IF P2M2_MachCtrl.U.DT_iMode=1 THEN
	D_Sys.bP2M2Enable:=TRUE;	
ELSE
	D_Sys.bP2M2Enable:=FALSE;
END_IF

D_Sys.fM2MainSetPos:=arrAxis[P2M2_Axise.VirAxisName.VirMain].NcToPlc.ActPos;//2号叠片主虚轴位置 20240509 CF
D_Pro.bAn_M2LockReady:=P2M2_MachCtrl.An_b.GetPiceReady;//正极取流水线极片准备好
D_Pro.bAn_M2JumpReady:=P2M2_MachCtrl.An_b.JumpPiceReady  OR (bDiffVel[2] AND NOT P2M2_MachCtrl.An_b.GetPiceReady);//正极跳过取流水线极片准备好 20240509 CF
D_Pro.bCa_M2LockReady:=P2M2_MachCtrl.Ca_b.GetPiceReady;//负极取流水线极片准备好
D_Pro.bCa_M2JumpReady:=P2M2_MachCtrl.Ca_b.JumpPiceReady;//负极跳过取流水线极片准备好
D_Pro.bAn_M2PoleHave:=P2M2_MachCtrl.An_b.bAn_PoleHave;
D_Pro.bCa_M2PoleHave:=P2M2_MachCtrl.Ca_b.bCa_PoleHave;
//模切给叠片的信号
P2M2_MachCtrl.An_b.An_MainBeltOK:=M_Pro.bAn_M2Allow;//允许正极取极片
P2M2_MachCtrl.Ca_b.Ca_MainBeltOK:=M_Pro.bCa_M2Allow;//允许负极取极片



//运行时间统计
	DT2_Timedata(
							Alm:=P2M2_DTSysState.bErrorStop AND NOT P2M2_DError AND NOT P2M2_MachCtrl.DT_b.DT_GMchange(*OR  P2M2_WJSysState.bErrorStop*) , 
							Wait:=P2M2_MachCtrl.U.DT_iMode=3 AND NOT P2M2_MachCtrl.DT_b.DT_GMchange AND (NOT P2M2_DTSysState.bErrorStop OR P2M2_DError (*AND NOT  P2M2_WJSysState.bErrorStop*) )  , 
							Run:= P2M2_MachCtrl.U.DT_iMode=1 (*AND P2M2_MachCtrl.U.WJ_iMode=1 AND P2M2_MachCtrl.U.TJ_iMode=1*), 
							Overhang_NG:= P2M2_MachCtrl.DT_b.DT_OverhangNG, 
							GM_change:=P2M2_MachCtrl.DT_b.DT_GMchange , 
							Query:=P2M2_MachCtrl.DT_b.Query, 
							date1:=P2M2_MachCtrl.DT_b.date1 , 								
							STTimedata=> );

							
							
//隔膜物料码OK
IF  (P3_PLC_PC_MES.Mes_PcToPlc6 AND  LEN(P3_PLC_PC_MES.Station2_Code)>6  ) OR P2M2_MachCtrl.DT_b.PartNumberOff THEN
	P2M2_MachCtrl.DT_b.DiaphragmPartNumberOK:=TRUE;
ELSE
	P2M2_MachCtrl.DT_b.DiaphragmPartNumberOK:=FALSE;
END_IF
//蓝胶物料码OK
IF  (P3_PLC_PC_MES.Mes_PcToPlc9 AND  LEN(P3_PLC_PC_MES.Station2_BlueCode)>6  ) OR P2M2_MachCtrl.DT_b.PartNumberOff THEN
	P2M2_MachCtrl.DT_b.BluePartNumberOK:=TRUE;
ELSE
	P2M2_MachCtrl.DT_b.BluePartNumberOK:=FALSE;
END_IF



IF P2M2_MachCtrl.DT_b.DiaphragmPartNumberOK THEN//隔膜料号OK
	CellMemory[P2M2_MachCtrl.DT_b.DT_Memory].Station_Code :=P3_PLC_PC_MES.Station2_Code;	
ELSE
	CellMemory[P2M2_MachCtrl.DT_b.DT_Memory].Station_Code :='';	
END_IF
IF P2M2_MachCtrl.DT_b.BluePartNumberOK THEN//蓝胶料号OK
	CellMemory[P2M2_MachCtrl.DT_b.DT_Memory].Station_BlueCode :=P3_PLC_PC_MES.Station2_BlueCode;	
ELSE
	CellMemory[P2M2_MachCtrl.DT_b.DT_Memory].Station_BlueCode :='';	
END_IF


	
//物料码清理
//隔膜条码重新校验
DT2Code_MES[1](CLK:=arrCyCtrl[P2M2_CycNo.CylinderName.PoleInflationCy].Status.ONState  , Q=> );  
IF DT2Code_MES[1].Q THEN
	P2M2_MachCtrl.DT_b.DiaphragmPartNumberOK:=FALSE;
	P3_PLC_PC_MES.Station2_Code:='';
	P3_PLC_PC_MES.Mes_PcToPlc6:=FALSE;
END_IF	

//蓝胶条码重新校验						
DT2Code_MES[2](CLK:= P2M2_MachCtrl.DT_b.HMI_WinBtn[1] , Q=> );  
IF DT2Code_MES[2].Q THEN
	P2M2_MachCtrl.DT_b.BluePartNumberOK:=FALSE;
	P3_PLC_PC_MES.Station2_BlueCode:='';
	P3_PLC_PC_MES.Mes_PcToPlc9:=FALSE;
END_IF									

(*						
//物料码校验报警
IF NOT P2M2_MachCtrl.DT_b.DiaphragmPartNumberOK AND NOT P2M2_MachCtrl.DT_b.PartNumberOff THEN
	P2M2_MachCtrl.DT_b.Error[55]:=TRUE;//叠台隔膜物料码校验未通过，请重新校验物料码
END_IF
IF NOT P2M2_MachCtrl.DT_b.BluePartNumberOK AND NOT P2M2_MachCtrl.DT_b.PartNumberOff THEN
	P2M2_MachCtrl.DT_b.Error[56]:=TRUE;//叠台蓝胶物料码校验未通过，请重新校验物料码
END_IF							
*)							
							


IF P2Btn.P2M2_Autobtn THEN
    arrCyCtrl[163].Cmd.bOFF:=TRUE;	//2号叠台		隔膜接带平台除尘
    arrCyCtrl[163].Cmd.bON:=FALSE;
ELSE
   arrCyCtrl[163].Cmd.bON:=TRUE;
   arrCyCtrl[163].Cmd.bOFF:=FALSE;
END_IF

END_PROGRAM

// ---- P2POUs/POUS/P2M3_Auto.TcPOU
PROGRAM P2M3_Auto
VAR
	DT3Code_MES: ARRAY[1..10] OF R_TRIG;
END_VAR

// 3号叠台自动
P2M3_program(
	DTselect:=3 , 
	Sys_Control:=P2M3_sysControl , 
	Mach_Control:=P2M3_MachCtrl , 
	arrCyNo:=P2M3_CycNo , 
	AxiseNo:=P2M3_Axise ,
	TableNo:=P2M3_TableNo ,
	Par:=P2M3_Par ,
	CCD:=P2M3_CCD,
	Torque:=P2M3_Torque,
	iTargetTorqueTest=>iTargetTorque[3]);
	
	

//叠片给模切的信号
D_Pro.bAn_M3Done:=P2M3_MachCtrl.An_b.AN_BeltDone; //正极取流水线极片完成
D_Pro.bAn_M3Safety:=P2M3_MachCtrl.An_b.AN_BeltSafe;//正极取流水线安全位
D_Pro.bCa_M3Done:=P2M3_MachCtrl.Ca_b.Ca_BeltDone;//负极取水线极片完成
D_Pro.bCa_M3Safety:=P2M3_MachCtrl.Ca_b.Ca_BeltSafe;//负极取流水线安全位
//D_Sys.fM3MainSetPos:=arrAxisCtrl[VirAxisNo.P2M3_VirMain].Cmd.fSetPos;
//D_Sys.bP2M3Enable:=P2M3_MachCtrl.U.DT_ModelChees;

IF P2M3_MachCtrl.U.DT_iMode=1 THEN
	D_Sys.bP2M3Enable:=TRUE;	
ELSE
	D_Sys.bP2M3Enable:=FALSE;
END_IF


D_Sys.fM3MainSetPos:=arrAxis[P2M3_Axise.VirAxisName.VirMain].NcToPlc.SetPos;//3号叠片主虚轴位置 20240509 CF
D_Pro.bAn_M3LockReady:=P2M3_MachCtrl.An_b.GetPiceReady;//正极取流水线极片准备好
D_Pro.bAn_M3JumpReady:=P2M3_MachCtrl.An_b.JumpPiceReady  OR (bDiffVel[3] AND NOT P2M3_MachCtrl.An_b.GetPiceReady);//正极跳过取流水线极片准备好 20240509 CF
D_Pro.bCa_M3LockReady:=P2M3_MachCtrl.Ca_b.GetPiceReady;//负极取流水线极片准备好
D_Pro.bCa_M3JumpReady:=P2M3_MachCtrl.Ca_b.JumpPiceReady;//负极跳过取流水线极片准备好
D_Pro.bAn_M3PoleHave:=P2M3_MachCtrl.An_b.bAn_PoleHave;
D_Pro.bCa_M3PoleHave:=P2M3_MachCtrl.Ca_b.bCa_PoleHave;
//模切给叠片的信号
P2M3_MachCtrl.An_b.An_MainBeltOK:=M_Pro.bAn_M3Allow;//允许正极取极片
P2M3_MachCtrl.Ca_b.Ca_MainBeltOK:=M_Pro.bCa_M3Allow;//允许负极取极片


//运行时间统计
 DT3_Timedata(						
							Alm:=P2M3_DTSysState.bErrorStop AND NOT P2M3_DError AND NOT P2M3_MachCtrl.DT_b.DT_GMchange(*OR  P2M3_WJSysState.bErrorStop*) , 
							Wait:=P2M3_MachCtrl.U.DT_iMode=3 AND NOT P2M3_MachCtrl.DT_b.DT_GMchange AND (NOT P2M3_DTSysState.bErrorStop OR P2M3_DError (*AND NOT  P2M3_WJSysState.bErrorStop*) )  , 
							Run:= P2M3_MachCtrl.U.DT_iMode=1 (*AND P2M3_MachCtrl.U.WJ_iMode=1 AND P2M3_MachCtrl.U.TJ_iMode=1*), 
							Overhang_NG:= P2M3_MachCtrl.DT_b.DT_OverhangNG, 
							GM_change:=P2M3_MachCtrl.DT_b.DT_GMchange , 
							Query:=P2M3_MachCtrl.DT_b.Query, 
							date1:=P2M3_MachCtrl.DT_b.date1 , 								
							STTimedata=> );

							
//隔膜物料码OK
IF  (P3_PLC_PC_MES.Mes_PcToPlc7 AND  LEN(P3_PLC_PC_MES.Station3_Code)>6  ) OR P2M3_MachCtrl.DT_b.PartNumberOff THEN
	P2M3_MachCtrl.DT_b.DiaphragmPartNumberOK:=TRUE;
ELSE
	P2M3_MachCtrl.DT_b.DiaphragmPartNumberOK:=FALSE;
END_IF
//蓝胶物料码OK
IF  (P3_PLC_PC_MES.Mes_PcToPlc10 AND  LEN(P3_PLC_PC_MES.Station3_BlueCode)>6  ) OR P2M3_MachCtrl.DT_b.PartNumberOff THEN
	P2M3_MachCtrl.DT_b.BluePartNumberOK:=TRUE;
ELSE
	P2M3_MachCtrl.DT_b.BluePartNumberOK:=FALSE;
END_IF



IF P2M3_MachCtrl.DT_b.DiaphragmPartNumberOK THEN//隔膜料号OK
	CellMemory[P2M3_MachCtrl.DT_b.DT_Memory].Station_Code :=P3_PLC_PC_MES.Station3_Code;	
ELSE
	CellMemory[P2M3_MachCtrl.DT_b.DT_Memory].Station_Code :='';	
END_IF
IF P2M3_MachCtrl.DT_b.BluePartNumberOK THEN//蓝胶料号OK
	CellMemory[P2M3_MachCtrl.DT_b.DT_Memory].Station_BlueCode :=P3_PLC_PC_MES.Station3_BlueCode;	
ELSE
	CellMemory[P2M3_MachCtrl.DT_b.DT_Memory].Station_BlueCode :='';	
END_IF


	
//物料码清理
//隔膜条码重新校验
DT3Code_MES[1](CLK:=arrCyCtrl[P2M3_CycNo.CylinderName.PoleInflationCy].Status.ONState  , Q=> );  
IF DT3Code_MES[1].Q THEN
	P2M3_MachCtrl.DT_b.DiaphragmPartNumberOK:=FALSE;
	P3_PLC_PC_MES.Station3_Code:='';
	P3_PLC_PC_MES.Mes_PcToPlc7:=FALSE;
END_IF	
//蓝胶条码重新校验	
				
DT3Code_MES[2](CLK:= P2M3_MachCtrl.DT_b.HMI_WinBtn[1] , Q=> );  
IF DT3Code_MES[2].Q THEN
	P2M3_MachCtrl.DT_b.BluePartNumberOK:=FALSE;
	P3_PLC_PC_MES.Station3_BlueCode:='';
	P3_PLC_PC_MES.Mes_PcToPlc10:=FALSE;
END_IF					

(*
//物料码校验报警
IF NOT P2M3_MachCtrl.DT_b.DiaphragmPartNumberOK AND NOT P2M3_MachCtrl.DT_b.PartNumberOff THEN
	P2M3_MachCtrl.DT_b.Error[55]:=TRUE;//叠台隔膜物料码校验未通过，请重新校验物料码
END_IF
IF NOT P2M3_MachCtrl.DT_b.BluePartNumberOK AND NOT P2M3_MachCtrl.DT_b.PartNumberOff THEN
	P2M3_MachCtrl.DT_b.Error[56]:=TRUE;//叠台蓝胶物料码校验未通过，请重新校验物料码
END_IF							
*)		





IF P2Btn.P2M3_Autobtn THEN
    arrCyCtrl[194].Cmd.bOFF:=TRUE;	///3号叠台		隔膜接带平台除尘
    arrCyCtrl[194].Cmd.bON:=FALSE;
ELSE
   arrCyCtrl[194].Cmd.bON:=TRUE;
   arrCyCtrl[194].Cmd.bOFF:=FALSE;
END_IF

END_PROGRAM

// ---- P2POUs/POUS/MAIN.TcPOU
PROGRAM MAIN
VAR
	rt:ARRAY[1..10]OF R_TRIG;//上升沿触发
	ft:ARRAY[1..10]OF F_TRIG;//下升沿触发
	i:BYTE;
	bSave: BOOL;
	rt10: R_TRIG;
	bReadDataFirstCyle: BOOL;
	testii: INT;
	testii2: INT;
	bSaveDataTest: BOOL;
	bReadDataCyle2: BOOL;
	rtSaveData: R_TRIG;
	fbDataXML  :FB_DataXML; 	
	
	
	
	BUSY: BOOL;
	ERR: BOOL;
	ERRID: UDINT;
	CSData:    CS_Data;
	

	THNN: INT;
	MA100: BOOL;
	A1: BOOL;
	D1: BOOL;
	A2: BOOL;
	A3: BOOL;
	
	//iShort:        IShortTest;
	D2: INT;
	//stTime: TIMESTRUCT;
	strTime: STRING;
	BY1:  BYTE;
	AA1: BOOL;
	btest: BOOL;
	iPower: INT;
	iPowerSetp: INT;
	bytePower: BYTE:=16#01;
	boPower2: BOOL;
	k: INT:=1;
	PowerOnDone: BOOL;
   
	SJ0617: INT;
	tRead										:TON;
END_VAR

VAR
	bFirstCycle										        	:BOOL;	(*初始化用的*)
(*保存掉电保持参数*)
	FB_WritePersistentData1								: FB_WritePersistentData;
	tCycleTimer											: TON;
	bWrite												: BOOL;    (*定时自动保存*)
(*系统重启*)
	tNtDelayReset										:TON;
	bReboot											: BOOL;	(*重启系统的变量*)
	NT_Reboot1											: NT_Reboot;
(*系统关机*)
	NT_Shutdown1										: NT_Shutdown;
	tNtDelayShutdown									: TON;
	bShutdown											: BOOL;
(*远程桌面接管*)
	OpenRemoteDesktop									: NT_StartProcess;
	timerHMI											:TON;
(*系统时间获取*)
	NT_GetTime1											: NT_GetTime;
(*心跳信号*)
	bHeartBeat											:BOOL;
	tHeartBeatTime										:TIME:=t#0.5s;
	TonHeartBeat										:TON;

	TaskInfo											:	TaskInfoCtrl;
	loadParaStep: UINT;

    tonPowerOn  :Tc2_Standard.TON;
    tonPower       :Tc2_Standard.TON;


     STR1: STRING:='20200412160000';
	 STR2: STRING:='12345678ABCDE';
	 STR3: STRING:='SSDDFF1234  JJJJ';
	 size:UDINT;
END_VAR

(*===========================================版本号=================================================*)
//MachimeVersion:='V3.0-24/3/2';(*HMI显示当前程序版本号*)
IF versionwrite THEN
   MachimeVersion:=CONCAT(CONCAT(CONCAT(CONCAT('V',CONCAT( WORD_TO_STRING(stTime.wYear),'.')),WORD_TO_STRING(stTime.wMonth)),'.'),WORD_TO_STRING(stTime.wDay));
END_IF
(*
版本： 


(*
1、线扫OK与NG信号IO触发;（02.20）
2、叠台NG梯度踢废空叠隔膜程序；（02.20）
3、叠台NG梯度踢废下料方式程序；（02.20）
4、隔膜剩余长度计算程序;（02.21）
5、无极片编号传送带尾部排废程序；（02.23）
6、对齐度NG计数程序  （02.27）
7、接带后找极耳程序；（02.28）
8、模切风刀吹气程序；（3.2）
9、程序版本号程序；（3.2）
10、叠台搬运极耳真空检测程序；（3.3）
11、冷压扫二维码程序；（3.3）
12、隔膜剩余长度计算（通过卷径大小）程序;（03.3）
13、隔膜卷径报警值限定（93），卷径报警实时判断改为叠完一个电芯判断一次;（03.6）
14、叠台搬运和压刀凸轮曲线修改，压刀升降和压刀开合行程限定；（03.12）
15、模切线扫结果判定逻辑优化，线扫触发和结果计数；（03.12）
16、新增模切放卷尾料4连标程序；（03.13）
17、模切黄标和接带踢废程序优化；（03.13）
18、短卷针回零增加安全条件(短卷针旋转轴原点传感器需亮)；（03.13）
19、模切放卷激光器继电器控制启用；（3.17）
20、触摸屏门禁屏蔽取消；（3.17）
21、增加启动CCD自检弹窗，需要确认后才能启动；（3.26）
22、叠台气涨轴开关有信号，隔膜踢废；（3.26）
23、触摸屏三级权限；（3.26）
24、上位机优率表；（3.31）
25、黄标跳切计数；（3.26）
26、黄标计数；（4.1）
27、叠台增加调试模式；（4.2）
28、热切丝寿命计数；（4.2）
29、模切尾料四连标检测；（4.2）
30、对齐度单片踢废；（4.5）
31、隔膜尾料角度计算；（4.5）
32、断带后R角不冲切；（4.7）
33、黄标与接带感应后日志；（4.7）
34、极片间距报警；（4.17）
35、凸轮位置角度固定；（4.17）
36、空叠首尾层隔膜降速降张力；（4.17）
37、正极真空改成常开；（4.17）
38、纠偏台重复精度测试；（4.17）
39、二维码贴胶完成自动备胶默停、重胶；（4.20）
40、对齐度踢废后第一片纠偏平台不纠偏；（4.20）
41、叠台一键初始化；（4.20）
42、模切尺寸、倒装、分段皮带比例系数改成一致；（4.20）
43、尾卷纠偏到限位，凸轮耦合报警；（4.20）
44、叠最后一层隔膜负极叠台升降放片位置下降少一点；（4.20）
45、模切R角横深纵深闭环纠偏；（4.20）
46、CCD标定与重复精度测试电机到位后延时拍照；（4.20）
47、短卷针夹泄气真空；（4.21）
48、对齐度闭环纠偏；（4.21）
49、模切触发高速停止；（4.22）
50、叠片取分段皮带取料中信号提前复位；（4.22）
51、贴胶头进退增加软限位；（4.23）
52、叠台0步增加判断，正负极不能执行同时往叠台方向运动流程；（4.23）
53、热压一键初始化；（4.23）
*)
*)
(*====================================================================================================*)

TwinCAT_Nt();
IF tonPowerOn.ET>=T#1S THEN
     MAIN.RecipeData();
END_IF
IOLink();

tonPowerOn(IN:=PowerOnDone , PT:=T#15S , Q=> , ET=> );  //上电延时5S

IF tonPowerOn.Q AND fbDataXML.bReadParDone THEN
  MainState();
  FingerprintKey();  
  dDrauFan[1];// :=TRUE;
  dDrauFan[2];// :=TRUE;
ELSE
   Power();//接触器上电
END_IF
op();



SJ0617;


//字体设置成中文字体  解决了注释乱码的问题






// scRecipe(iRecipe2:=iRecipe );

ACTION op:
FOR i :=1 TO 50 DO
	IF Network1_OP[i] = 8 THEN
		bNetwork1_OP[i] := TRUE;
	ELSE
		bNetwork1_OP[i] := FALSE;
	END_IF
	
	IF Network2_OP[i] = 8 THEN
		bNetwork2_OP[i] := TRUE;
	ELSE
		bNetwork2_OP[i] := FALSE;
	END_IF
	
	IF Network3_OP[i] = 8 THEN
		bNetwork3_OP[i] := TRUE;
	ELSE
		bNetwork3_OP[i] := FALSE;
	END_IF
	
	IF Network4_OP[i] = 8 THEN
		bNetwork4_OP[i] := TRUE;
	ELSE
		bNetwork4_OP[i] := FALSE;
	END_IF
	
	IF Network5_OP[i] = 8 THEN
		bNetwork5_OP[i] := TRUE;
	ELSE
		bNetwork5_OP[i] := FALSE;
	END_IF
END_FOR
END_ACTION

ACTION Power:
(***系统延时启动***)

tonPower(IN:= , PT:=T#1.5S , Q=> , ET=> );

CASE iPowerSetp OF
0:
    tonPower.IN:=TRUE;
    iPowerSetp:=10;
10:
   IF   tonPower.Q  THEN
      bytePower:=SHL(bytePower,1);
     
      tonPower(IN:=FALSE );
      k:=k+1;
     iPowerSetp:=20;
  END_IF
20:
    bytePower.0:=1;
    tonPower.IN:=TRUE;
    iPowerSetp:=30;
30:
   IF  k>=8 THEN
        iPowerSetp:=666;
       // bytePower:=16#00;
        PowerOnDone:=TRUE;
   ELSE
      iPowerSetp:=10;
   END_IF

END_CASE
 
bytePower.0;
bytePower.1;
bytePower.2;
bytePower.3;
bytePower.4;
bytePower.5;
bytePower.6;
bytePower.7;
END_ACTION

ACTION RecipeData:

IF NOT  bReadDataFirstCyle AND tCycleTimer.ET>T#90S THEN //testii:=testii+1
	//fbDataXML.bRead:=NOT bDataValid;
	bReadDataFirstCyle:=TRUE;
END_IF


IF fbDataXML.bReadParDone AND bReadDataFirstCyle AND NOT  bReadDataCyle2 THEN
	  parDA:=P2User1_Par.parDA;
	  parFilterAD:=P2User1_Par.parFilterAD;//  先备份数据暂时不开放 
      bReadDataCyle2:=TRUE;
END_IF

rt[2](CLK:=tCycleTimer.ET>=T#4M , Q=> );
rtSaveData(CLK:=stHmiSysCmd.bSaveData , Q=> );
IF  rtSaveData.Q THEN
	bSaveDataTest:=TRUE;
END_IF
IF  rt[2].Q  OR  bSaveDataTest THEN   
	P2User1_Par.parDA:=parDA;
	P2User1_Par.parFilterAD:=parFilterAD; 
	bSaveDataTest:=FALSE;
	fbDataXML.bSave:=TRUE;
	testii2:=testii2+1;
END_IF

rt[4](CLK:=stHmiSysCmd.bReadData (*AND P2M1_MachCtrl.U.DT_iMode=3 AND P2M2_MachCtrl.U.DT_iMode=3 AND P2M3_MachCtrl.U.DT_iMode=3*), Q=> );
rt[5](CLK:=PowerOnDone , Q=> );
tRead(IN:=PowerOnDone, PT:=T#3S , Q=> , ET=> );
IF PowerOnDone AND  tRead.Q AND NOT fbDataXML.bReadParDone THEN
	 P2M3_MachCtrl.DT_b.Error[67]:=TRUE;//上电后叠台参数读取失败，请手动点读取参数
END_IF

fbDataXML(
					bSave:=fbDataXML.bSave AND NOT P2M3_MachCtrl.DT_b.Error[67] , 
					bRead:=fbDataXML.bRead OR rt[5].Q OR rt[4].Q , 
					bSaveParDone=> , 
					bReadParDone=> );

fbDataXML.bSaveParDone;
fbDataXML.bReadParDone;


(*
tCycleTimer(IN:=NOT tCycleTimer.Q , PT:=T#300S , Q=>bSave , ET=> );
rt10(clk:=bSave);
IF NOT  bReadDataFirstCyle THEN //testii:=testii+1
	 fbDataXML.bRead:=TRUE;
	 testii:=testii+1;
	 bReadDataFirstCyle:=TRUE;
END_IF


IF fbDataXML.bReadParDone AND bReadDataFirstCyle AND NOT  bReadDataCyle2 THEN
	  //parDA:=P2User1_Par.parDA;
	  //parFilterAD:=P2User1_Par.parFilterAD;      //  先备份数据暂时不开放 
      bReadDataCyle2:=TRUE;
END_IF


rtSaveData(CLK:=stHmiSysCmd.bSaveData , Q=> );
IF  rtSaveData.Q THEN
	bSaveDataTest:=TRUE;
END_IF


IF  rt10.Q   OR   bSaveDataTest THEN
   
     P2User1_Par.parDA:=parDA;
	 P2User1_Par.parFilterAD:=parFilterAD; 

    bSaveDataTest:=FALSE;

	fbDataXML.bSave:=TRUE;
	testii2:=testii2+1;
END_IF

fbDataXML(bSave:=fbDataXML.bSave AND M_Sys .P1SaveParDone , 
                      bRead:=fbDataXML.bRead AND M_Sys.P1ReadParDone ,
                      bSaveParDone=> , 
                      bReadParDone=>,);
(*
IF fbDataXML.bError THEN				  
		P3_Error[91]:=TRUE;	
END_IF			
*)	 					   
P2SaveParDone:=fbDataXML.bSaveParDone;
P2ReadParDone:=fbDataXML.bReadParDone;
*)
END_ACTION

ACTION TwinCAT_Nt:
//fPlcCycleTime_ms:=UDINT_TO_LREAL(_TaskInfo[0].CycleTime)/10000;

(***********************  保存掉电保持数据   **************************************)
tCycleTimer(IN:=NOT tCycleTimer.Q , PT:=T#386S , Q=>bWrite , ET=> );
rt[1](CLK:=tCycleTimer.ET>=T#3M, Q=>bWrite );
FB_WritePersistentData1(
	NETID:='' ,
	PORT:=852 ,
	START:=bWrite OR  stHmiSysCmd.bSaveData   ,//OR    _TaskInfo[1].FirstCycle
	TMOUT:=t#2s ,
	MODE:=SPDM_2PASS ,
	BUSY=>BUSY ,
	ERR=> ERR,
	ERRID=>ERRID );
ft[1](CLK:=BUSY , Q=> );
IF ft[1].Q THEN
	bDataValid:=TRUE;
END_IF	
	
(********************** 获取系统时间   ***************************************)
NT_GetTime1(
	NETID:='' ,
	START:=Pulse._1s.RT ,
	TMOUT:= ,
	BUSY=> ,
	ERR=> ,
	ERRID=> ,
	TIMESTR=>stTime );

	strTime:=CONCAT(CONCAT(CONCAT(CONCAT(CONCAT(CONCAT(CONCAT(CONCAT( CONCAT(CONCAT( WORD_TO_STRING(stTime.wYear),'-'), WORD_TO_STRING(stTime.wMonth)),'-'),WORD_TO_STRING(stTime.wDay)),
             '-'),WORD_TO_STRING(stTime.wHour)),'-'),WORD_TO_STRING(stTime.wMinute)),'-'),WORD_TO_STRING(stTime.wSecond));

(********************************** Systemfunctions **********************************************************)
	SysInfo(
		Reset				:= ,
		TimeStampTrig		:= Pulse._100ms.RT,
		//RunTimeNo			=> ,
		//ProjectName			=> ,
		//NumberOfTasks		=> ,
		//OnlineChangeCount	=> ,
		RetainVarErr		=> ,
		PersistenVarErr		=> ,
		TimeStampDT			=> ,
		TimeStamp			=> ,
		TimeStr				=> ,
		DateStr				=> ,
		TimeStamp2			=> ,
		TimeStruct			=> ,
		MonthDays			=> ,
		LeapYear			=> ,
		WeekOfYear			=> ,
		timezoneId			=>);

	TaskInfo(
		index				=> ,
		active				=> ,
		taskName			=> ,
		firstCycle			=> ,
		cycleTimeExceeded	=> ,
		cycleTime			=> ,
		lastExecTime		=> ,
		priority			=> ,
		cycleCount			=> );

	Pulse(
		BlinkSlow			=> ,
		Blink				=> ,
		BlinkFast			=> );	
		
	(*系统重启，CE远程桌面，系统时间，定时保存掉电数据，等系统常规动作*)
(**********************  通讯心跳信号   ***************************************)
TonHeartBeat(IN:=NOT TonHeartBeat.Q , PT:=tHeartBeatTime , Q=> , ET=> );
IF TonHeartBeat.Q THEN
	bHeartBeat:=NOT bHeartBeat;
END_IF

tNtDelayReset(IN:=stHmiSysCmd.bRebootPc OR bReboot , PT:=T#1S , Q=> , ET=> );
NT_Reboot1(
	NETID:='' ,
	DELAY:= ,
	START:=tNtDelayReset.Q  ,
	TMOUT:=DEFAULT_ADS_TIMEOUT ,
	BUSY=> ,
	ERR=> ,
	ERRID=> );

tNtDelayShutdown(IN:=stHmiSysCmd.bShutDownPc OR bShutDown , PT:=T#1S , Q=> , ET=> );	(*触摸屏上已经做了延时*)
NT_Shutdown1(
	NETID:= ,
	DELAY:= ,
	START:=tNtDelayShutdown.Q,
	TMOUT:=DEFAULT_ADS_TIMEOUT ,
	BUSY=> ,
	ERR=> ,
	ERRID=> );
END_ACTION

END_PROGRAM

// ---- P2POUs/BasicFunction/08_Data/FB_DataXML.TcPOU
FUNCTION_BLOCK FB_DataXML
VAR_INPUT
    	bSave:BOOL;
	    bRead:BOOL;
		bReadSel:BOOL;//参数读取选择，TRUE=选择恢复上电备份的参数
END_VAR
VAR_OUTPUT
    	bSaveParDone      :BOOL;
	    bReadParDone     :BOOL;
END_VAR

VAR
	iDataSetp: INT;
	i1: INT;
	i2:BYTE;
	rt100:Tc2_Standard.R_TRIG;
	rt101:Tc2_Standard.R_TRIG;
	rt102:Tc2_Standard.R_TRIG;
	rt103:Tc2_Standard.R_TRIG;
	bSaveTemp: BOOL;
	bReadTemp: BOOL;
	sFilePath:STRING;//文件路径
	sNewFilePath:STRING;//新文件路径
	sOldFilePath:STRING;//旧文件路径
	sFileName:STRING;//文件名称
	sVarName:STRING;//变量名称
	fbXmlSrvRead				: FB_XmlSrvReadByName;//读取XML文件	
	fbXmlSrvWrite				: FB_XmlSrvWriteByName;//写入XML文件
	bFirstCycleFlg:BOOL;//首次执行标志位
	fbGetFileList: FB_GetFileList;//获取文件列表功能块
	stFindFileEntry:ARRAY[1..50] OF ST_FindFileEntry;//文件列表存放结构体	
	nFileBakStep:UINT;//文件备份步序
	fbFileDelete	: FB_FileDelete;//删除文件
	fbFileRename	: FB_FileRename;//文件重命名
	fbCreateDirectory:FB_CreateDirectory;//文件夹创建
END_VAR

M_WriteOrRead();
A_FileBak();

ACTION A_FileBak:
CASE nFileBakStep OF
	200:
		fbGetFileList(bExecute:=FALSE);
		fbFileDelete(bExecute:=FALSE);
		fbFileRename(bExecute:=FALSE);
		fbCreateDirectory(bExecute:=FALSE);
		nFileBakStep:=300;
	300:(*获取文件列表*)
		fbGetFileList.pFindFileListADR:=ADR(stFindFileEntry);
		fbGetFileList.u32FindFileListSizeOf:=SIZEOF(stFindFileEntry);
		fbGetFileList(bExecute:=TRUE,sgPathName:=sOldFilePath,sgFileType:='xml');	
		IF fbGetFileList.bDone THEN
			fbGetFileList(bExecute:=FALSE);
			nFileBakStep:=310;
		ELSIF fbGetFileList.bError THEN
			fbGetFileList(bExecute:=FALSE);
			nFileBakStep:=997;
		END_IF
	310:(*判断文件是否存在，文件存在则备份一次，文件不存在直接给完成信号*)
		FOR i2:=1 TO 50 DO
			IF stFindFileEntry[i2].sFileName=sFileName THEN//
				EXIT;
			END_IF
		END_FOR
		IF i2>50 THEN
			nFileBakStep:=666;
		ELSE
			nFileBakStep:=320;
		END_IF
	320:(*文件夹创建*)
	fbCreateDirectory(bExecute:=TRUE , sgPathName:=sNewFilePath, tTimeout:=T#1S );
	IF fbCreateDirectory.bDone THEN
		fbCreateDirectory(bExecute:=FALSE);
		nFileBakStep:=350;
	ELSIF fbCreateDirectory.bError THEN
		fbCreateDirectory(bExecute:=FALSE);
		nFileBakStep:=998;
	END_IF
	350:(*删除旧文件*)
		fbFileDelete.sPathName:= CONCAT(sNewFilePath,sFileName);
		fbFileDelete(bExecute:=TRUE,ePath:= PATH_GENERIC,tTimeout:=T#5S);
		IF NOT fbFileDelete.bBusy THEN
			fbFileDelete(bExecute:=FALSE);
			nFileBakStep:=360;
		END_IF
	360:(*重命名文件*)
		fbFileRename.sOldName:= CONCAT(sOldFilePath,sFileName);
		fbFileRename.sNewName:= CONCAT(sNewFilePath,sFileName);
		fbFileRename(bExecute:=TRUE,ePath:= PATH_GENERIC,tTimeout:=T#5S);
		IF NOT fbFileRename.bBusy THEN
			fbFileRename(bExecute:=FALSE);
			IF NOT fbFileRename.bError THEN
				nFileBakStep:=666;
			ELSE
				nFileBakStep:=999;
			END_IF			
		END_IF
END_CASE
END_ACTION

ACTION M_WriteOrRead:
rt100(CLK:=bSave , Q=> );//保存参数
rt101(CLK:=bRead , Q=> );//读取参数
IF rt100.Q THEN  //保存参数
    bSaveTemp:=TRUE;
	bReadTemp:=FALSE;
	bSaveParDone:=FALSE;
	iDataSetp:=50;
END_IF
IF rt101.Q THEN  //读取参数
    bReadTemp:=TRUE;
    bSaveTemp:=FALSE;
	bReadParDone:=FALSE;
	iDataSetp:=50;
END_IF

//rt102(CLK:=NOT bFirstCycleFlg AND NOT bReadTemp, Q=> );//首次上电自动备份参数
IF rt102.Q THEN  //首次上电自动备份参数
	iDataSetp:=50;
END_IF

CASE  iDataSetp OF 
	50:
		I1:=1;
		fbXmlSrvRead(bExecute:=FALSE);
		fbXmlSrvWrite(bExecute:=FALSE);
		bSave:=FALSE;
		bRead:=FALSE;
		iDataSetp:=100;
	 100:
	 	sFilePath:='C:\P2XML\';//保存文件路径
		CASE I1 OF 
			1://轴参数
				sFileName  := 'P2arrAxisPar.xml';
				sVarName:='GMotion.arrAxisPar';
		(*		
			2://iModeEN
				sFileName  := 'P2iModeEN.xml';
				sVarName:='GVL_Par.iModeEN';
	     *)
			2://P2M1_Par
				sFileName  := 'P2M1_Par.xml';
				sVarName:='GVL_Par.P2M1_Par';
			3://P2M2_Par
				sFileName  := 'P2M2_Par.xml';
				sVarName:='GVL_Par.P2M2_Par';
			4: //P2M3_Par 
				sFileName  := 'P2M3_Par.xml';
				sVarName:='GVL_Par.P2M3_Par';
			5: // P2User1_Par
				sFileName  := 'P2User1_Par.xml';
				sVarName:='GVL_Par.P2User1_Par';
				
			(*	
			7: // P2M1_Production
				sFileName  := 'DT1Data.xml';
				sVarName:='GVL_Par.P2M1_Production';
			8: // P2M2_Production
				sFileName  := 'DT2Data.xml';
				sVarName:='GVL_Par.P2M2_Production';
			9: // P2M3_Production
				sFileName  := 'DT3Data.xml';
				sVarName:='GVL_Par.P2M3_Production';
		
			10: // P2User1_Par
				sFileName  := 'FilterAD.xml';
				sVarName:='GVL_Par.P2User1_Par';
			*)	
		END_CASE
		IF  bSaveTemp THEN
			iDataSetp:=200;
		ELSIF  bReadTemp THEN
			iDataSetp:=300;	
		//ELSIF NOT bFirstCycleFlg THEN
		//	iDataSetp:=400;
		END_IF
		
	(********************保存数据流程：先备份原来参数再保存新参数，如果保存失败恢复至备份参数********************)
	200:(*开始备份*)
		sNewFilePath:=CONCAT(sFilePath,'Tmp\');
		sOldFilePath:=sFilePath;
		nFileBakStep:=200;//调用A_FileBak()进行文件备份
		iDataSetp:=210;
	210:(*文件备份状态判断*)
		IF nFileBakStep=666 THEN//文件备份成功，保存新参数
			iDataSetp:=230;
		ELSIF nFileBakStep>990 THEN//文件备份失败
			iDataSetp:=997;			
		END_IF
	230:(*保存新参数*)	
		fbXmlSrvWrite(
			bExecute:= TRUE, 
			ePath:=PATH_GENERIC , 
			nMode:=XMLSRV_ADDMISSING , 
			sSymName:=sVarName , 
			sFilePath:= CONCAT(sFilePath,sFileName), 
			sXPath:= '/DataEntry/Value', 
			tTimeout:= T#2S);
		IF NOT fbXmlSrvWrite.bBusy THEN
			fbXmlSrvWrite(bExecute:=FALSE);
			IF NOT fbXmlSrvWrite.bError THEN(*保存新参数成功*)
				iDataSetp:=500;
			ELSE(*保存新参数失败，恢复未写入新参数前的备份*)
				iDataSetp:=250;
			END_IF	
		END_IF
	250:(*保存新参数失败，恢复未写入新参数前的备份*)
		sOldFilePath:=CONCAT('Tmp\' ,sFileName);
		sNewFilePath:=sFilePath;
		nFileBakStep:=200;//调用A_FileBak()进行文件备份
		iDataSetp:=260;
	260:(*恢复文件状态判断*)
		IF nFileBakStep=666 THEN//文件恢复成功
			iDataSetp:=500;
		ELSIF nFileBakStep>990 THEN//文件恢复失败
			iDataSetp:=998;			
		END_IF		

	(********************参数读取流程********************)	
	300:(*参数读取选择，TRUE=选择恢复上电备份的参数*)
		IF bReadSel THEN
			sFilePath:=CONCAT(sFilePath,'Bak\');
		END_IF
		iDataSetp:=310;
	310:(*读取参数*)
		fbXmlSrvRead(
			bExecute:= TRUE, 
			ePath:=PATH_GENERIC , 
			nMode:=XMLSRV_ADDMISSING , 
			sSymName:= sVarName, 
			sFilePath:=CONCAT(sFilePath,sFileName) , 
			sXPath:='/DataEntry/Value' , 
			tTimeout:=T#2S);
		IF NOT fbXmlSrvRead.bBusy THEN
			fbXmlSrvRead(bExecute:=FALSE);
			IF NOT fbXmlSrvRead.bError THEN
				iDataSetp:=500;//读取成功
			ELSE
				iDataSetp:=999;//读取失败
			END_IF
		END_IF
		
	(********************上电自动备份流程，防止被覆盖********************)	
	400:
		sOldFilePath:=sFilePath;
		sNewFilePath:=CONCAT(sFilePath,'Bak\' );
		nFileBakStep:=200;//调用A_FileBak()进行文件备份
		iDataSetp:=410;
	410:
		IF nFileBakStep=666 THEN
				iDataSetp:=500;
		ELSIF nFileBakStep>990 THEN
				iDataSetp:=999;			
		END_IF
	500:(*继续写下个文件*)
		IF 1<=i1 AND i1<5 THEN
			i1:=i1+1; 
			iDataSetp:=100; 
		ELSIF i1>=5 THEN
			IF  bSaveTemp THEN		
				bSaveParDone:=TRUE;
			ELSIF  bReadTemp THEN
				bReadParDone:=TRUE;
			ELSIF NOT bFirstCycleFlg THEN
				bFirstCycleFlg:=TRUE;
			END_IF
			bReadSel:=FALSE;
			bReadTemp:=FALSE;
			bSaveTemp:=FALSE;
			iDataSetp:=666;   
		END_IF
END_CASE
END_ACTION

END_FUNCTION_BLOCK

// ---- P2POUs/BasicFunction/08_Data/CS_Data.TcPOU
FUNCTION_BLOCK CS_Data
VAR_INPUT
END_VAR
VAR_OUTPUT
END_VAR
VAR
	//tDataSave:TON;
	//fbSaveData:FB_WritePersistentData;
	//fbXMLWrite:FB_XMLSrvWrite;
	//bWriteXml: BOOL;
	
	fbFileOpen_w:fb_fileopen;
	//fbFileOpen_r:fb_fileopen;
	fbFileWrite:fb_filewrite;
	fbFileRead:FB_FileRead;
	fbFileClose_w:fb_FileClose;
	//fbFileClose_r:fb_FileClose;
	HFILE:UINT;
	//HFILE_R:UINT;
	//bFileOpen_w:BOOL;
	//bFileOpen_r:BOOL;
	//bFileWrite:BOOL;
	//bFileClose_w:BOOL;
	//bFileClose_r:BOOL;
	//bFileRead:BOOL;
	bSave:BOOL;
	bRead:BOOL;
//	tFileOper_Save:TON;
	//tFileOper_Read:TON;
	iDataSetp: INT;
	TON10:Tc2_Standard.TON;
	bExecute: BOOL;
	I1: INT;
	rt100:Tc2_Standard.R_TRIG;
	rt101:Tc2_Standard.R_TRIG;
	bExecute1: BOOL;
	bExecute2: BOOL;
	bExecute3: BOOL;	

	bSaveTemp: BOOL;
	bReadTemp: BOOL;
	bReadDataOk: BOOL;
END_VAR


M_WriteOrRead();

ACTION M_WriteOrRead:


(*
rt100(CLK:=bSave , Q=> );//保存参数
rt101(CLK:=bRead , Q=> );//读取参数

IF rt100.Q THEN
	iDataSetp:=100;
	TON10.IN:=FALSE;
	I1:=1;
	bExecute1:=FALSE;
	bExecute2:=FALSE;	
	bExecute3:=FALSE;	
	bSave:=FALSE;
	bRead:=FALSE;
    bSaveTemp:=TRUE;
	bReadTemp:=FALSE;
END_IF

IF rt101.Q THEN
	iDataSetp:=100;
	TON10.IN:=FALSE;
	I1:=1;
	bExecute1:=FALSE;
	bExecute2:=FALSE;	
	bExecute3:=FALSE;	
	bSave:=FALSE;
	bRead:=FALSE;
    bReadTemp:=TRUE;
    bSaveTemp:=FALSE;
END_IF

TON10(IN:= , PT:=T#200MS , Q=> , ET=> );
//保存配方	
CASE  iDataSetp OF 
	
	100:	//参数给定
	   
	   IF bSaveTemp THEN
	     fbFileOpen_w.nMode:=FOPEN_MODEWRITE OR FOPEN_MODEBINARY;
	   END_IF
	   IF bReadTemp THEN
	     fbFileOpen_w.nMode:=FOPEN_MODEREAD OR  FOPEN_MODEBINARY;
	   END_IF
	  iDataSetp:=101;
	101:

	  CASE I1 OF 
		1:
		 fbFileWrite.pWriteBuff:=ADR(gstM1Par);
		 fbFileWrite.cbWriteLen:=SIZEOF(gstM1Par);
		 fbFileRead.pReadBuff:=ADR(gstM1Par1);
		 fbFileRead.cbReadLen:=SIZEOF(gstM1Par1);
		 fbFileOpen_w.sPathName:='C:\P2Data\M1.bin';
		2:
		 fbFileWrite.pWriteBuff:=ADR(gstM2Par);
		 fbFileWrite.cbWriteLen:=SIZEOF(gstM2Par);
		 fbFileRead.pReadBuff:=ADR(gstM2Par1);
		 fbFileRead.cbReadLen:=SIZEOF(gstM2Par1);
		 fbFileOpen_w.sPathName:='C:\P2Data\M2.bin';
		3:
		 fbFileWrite.pWriteBuff:=ADR(gstM3Par);
		 fbFileWrite.cbWriteLen:=SIZEOF(gstM3Par);
		 fbFileRead.pReadBuff:=ADR(gstM3Par1);
		 fbFileRead.cbReadLen:=SIZEOF(gstM3Par1);
		 fbFileOpen_w.sPathName:='C:\P2Data\M3.bin';
		4:
		 fbFileWrite.pWriteBuff:=ADR(gstM4Par);
		 fbFileWrite.cbWriteLen:=SIZEOF(gstM4Par);
		 fbFileRead.pReadBuff:=ADR(gstM4Par1);
		 fbFileRead.cbReadLen:=SIZEOF(gstM4Par1);
		 fbFileOpen_w.sPathName:='C:\P2Data\M4.bin';
		5:  
		 fbFileWrite.pWriteBuff:=ADR(gstM5Par);
		 fbFileWrite.cbWriteLen:=SIZEOF(gstM5Par); 
		 fbFileRead.pReadBuff:=ADR(gstM5Par1);
		 fbFileRead.cbReadLen:=SIZEOF(gstM5Par1);
		 fbFileOpen_w.sPathName:='C:\P2Data\M5.bin';
	  END_CASE
	  iDataSetp:=200;
	
	200:	//打开文件
		bExecute1:=TRUE;
		TON10.IN:=TRUE;
	  IF TON10.Q THEN
		 bExecute1:=FALSE; 
		 TON10.IN:=FALSE;
		 iDataSetp:=300; 
	  END_IF
	
	300:	//读写文件
		bExecute2:=TRUE;
		TON10.IN:=TRUE;
	  IF TON10.Q THEN
		  bExecute2:=FALSE; 
		  TON10.IN:=FALSE;
		 iDataSetp:=400; 
	  END_IF
	
	400:	//关闭文件
		bExecute3:=TRUE;
		TON10.IN:=TRUE;
	  IF TON10.Q THEN
		  bExecute3:=FALSE; 
		  TON10.IN:=FALSE;
		  iDataSetp:=500; 
	  END_IF
	
	500://继续写下个文件
	  IF I1>=1 AND I1<5 THEN
		 I1:=I1+1; 
		 TON10.IN:=FALSE;
		 iDataSetp:=100; 
		 bExecute1:=FALSE; 
		 bExecute2:=FALSE; 
		 bExecute3:=FALSE; 
	  ELSIF I1>=5 THEN
		  bReadTemp:=FALSE;
          bSaveTemp:=FALSE;
		 iDataSetp:=666;   
	  END_IF
END_CASE


IF bReadDataOk THEN
   gstM1Par:=gstM1Par1;
   gstM2Par:=gstM2Par1;
   gstM3Par:=gstM3Par1;
   gstM4Par:=gstM4Par1;	
   gstM5Par:=gstM5Par1;
   bReadDataOk:=FALSE;
END_IF










   	fbFileOpen_w(
	sNetId:= , 
	sPathName:= , //C:\P2Data
	nMode:=   , 
	ePath:=PATH_GENERIC , 
	bExecute:=bExecute1 , 
	tTimeout:=T#3S , 
	bBusy=> , 
	bError=> , 
	nErrId=> , 
	hFile=>hfile );


	fbFileWrite(
	sNetId:= , 
	hFile:= hFile, 
	pWriteBuff:= , 
	cbWriteLen:= , 
	bExecute:=bExecute2 AND bSaveTemp, 
	tTimeout:=T#3S , 
	bBusy=> , 
	bError=> , 
	nErrId=> , 
	cbWrite=> );



	fbFileRead(
	sNetId:= , 
	hFile:=hFile , 
	pReadBuff:= , 
	cbReadLen:= , 
	bExecute:= bExecute2 AND bReadTemp, 
	tTimeout:= T#3S, 
	bBusy=> , 
	bError=> , 
	nErrId=> , 
	cbRead=> , 
	bEOF=> );


	fbFileClose_w(
	sNetId:= , 
	hFile:= hFile, 
	bExecute:= bExecute3, 
	tTimeout:=T#3S , 
	bBusy=> , 
	bError=> , 
	nErrId=> );
	
	
	
*)
END_ACTION

END_FUNCTION_BLOCK

// ---- P2POUs/BasicFunction/11_SystemInfo/TaskInfoCtrl.TcPOU
FUNCTION_BLOCK TaskInfoCtrl
VAR_INPUT
END_VAR
VAR_OUTPUT
	index						:	INT;
	active					:	BOOL; 		(* Diese Variable zeigt an, ob die Task aktiv ist.*)
	taskName					:	STRING(16);	(* Der Taskname.*)
	firstCycle				:	BOOL;			(* Diese Variable hat im ersten Zyklus der SPS-Task den Wert: TRUE.*)
	cycleTimeExceeded		:	BOOL;			(* In dieser Variablen wird ein 躡erschreiten der eingestellten Taskzykluszeit gemeldet*)
	cycleTime				:	UDINT;		(* Eingestellte Taskzykluszeit in Vielfachen von 100ns*)
	lastExecTime			:	UDINT;		(* Ben鰐igte Zykluszeit f黵 den letzten Zyklus in Vielfachen von 100 ns*)
	MaxExecTime				:	UDINT;		(* Maximale Zykluszeit *)
	priority					:	BYTE;			(* Eingestellte Prioritaet der Task*)
	cycleCount				: 	UDINT;		(* Zykluszaehler*)
END_VAR

VAR
	GETCURTASKINDEX		: GETCURTASKINDEX;
END_VAR

	(*********************************************************************************)
	(*	(c) by Beckhoff Automation																		*)
	(*																											*)
	(*		B E C K H O F F   N E W   A U T O M A T I O N   T E C H N O L O G Y        *)
	(*																											*)
	(*		Eiserstr.5	D-33415 Verl	Germany	phone:	+49-5246-0	www.Beckhoff.com	*)
   (*																											*)
   (*		Bausteinbeschreibung	: Auswerten des SystemInfoTaskArrays 						*)
	(*																											*)
	(*		Version				:	V1.0																	*)
	(*		Stand					:	04.2009																*)
 	(*		Autor					:	Daniel Schlingmann												*)
	(*																											*)
	(*********************************************************************************)

(* Get Current Task Index ************************************************************************)
	GETCURTASKINDEX(index => index);

	(* Retein/Persisten Data Err *)
	//active :=  _TaskInfo[index].active;
	taskName :=  _TaskInfo[index].TaskName;
	firstCycle :=  _TaskInfo[index].FirstCycle;
	cycleTimeExceeded :=  _TaskInfo[index].CycleTimeExceeded;
	cycleTime :=  _TaskInfo[index].CycleTime;
	lastExecTime :=  _TaskInfo[index].LastExecTime;
	MaxExecTime	:= MAX(lastExecTime,MaxExecTime);
//	priority :=  _TaskInfo[index].Priority;
	firstCycle :=  _TaskInfo[index].FirstCycle;
	cycleCount :=  _TaskInfo[index].CycleCount;

(**************************************************************************************************)

END_FUNCTION_BLOCK

// ---- P2POUs/POUS/IOLink.TcPOU
PROGRAM IOLink
VAR
//	tFlash: TON;
//	bFlash:BOOL;
//	bIOinit: BOOL;
	XXX: INT;
	Q20815: BOOL;
	AA: INT;

     arrFilter_AD               : ARRAY[1..MaxAINo]  OF  FB_Filter_AD ;
      arrFilter_ADV2               : ARRAY[1..3]  OF  FB_Filter_ADV2 ;


    Test:BOOL;
	I1: INT;

    rt01   :Tc2_Standard.R_TRIG;
    rt02   :Tc2_Standard.R_TRIG;

     parDAOld                   :ARRAY[1..44] OF INT;   
	 q:INT;


END_VAR

P2_InPut();

P2_OutPut();

AI();

//LimitSwitch();

P2_AutoLink();
P2M1_AutoLink();
P2M2_AutoLink();
P2M3_AutoLink();
LimitSwitch();


IF fbPulseCtrl[4].RT THEN
      AO();
END_IF
(*
//rt01(CLK:=arrCyCtrl[P3CYNo.RollPress].Cmd.bON , Q=> );
//rt02(CLK:=arrCyCtrl[P3CYNo.RollPress].Cmd.bOFF , Q=> );
IF rt01.Q THEN
    P3EL4004S[3,1]:=parDA[33]	 ;//重力补偿
  //  P3EL4004S[3,2]:=parDA[34]	 ;
END_IF
IF rt02.Q THEN
    P3EL4004S[3,1]:=22000;//重力补偿
 //   P3EL4004S[3,2]:=20000;
END_IF



*)





AA;

ACTION AI:
//1号叠片
arrFilter_AD[1].AD	:=AI30[1];	//1号叠片	隔膜卷径超声波检测
arrFilter_AD[1].iMode:=2;
arrFilter_AD[1].fPointNum:=20;

arrFilter_AD[2].AD	:=AI30[2];	//1号叠片	隔膜放卷纠偏前检测
arrFilter_AD[2].iMode:=2;
arrFilter_AD[2].fPointNum:=20;//30;

arrFilter_AD[3].AD	:=AI30[3];	//1号叠片	隔膜放卷纠偏后检测
arrFilter_AD[3].iMode:=2;
arrFilter_AD[3].fPointNum:=20;//30;

//arrFilter_AD[4].AD	:=AI30[4];//1号叠片	隔膜张力检测
arrFilter_ADV2[1].AD	:=AI30[4];//1号叠片	隔膜张力检测
arrFilter_ADV2[1].iMode:=2;
arrFilter_ADV2[1].fPointNum:=1000;
//2号叠片
arrFilter_AD[5].AD	:=ABS(AI40[1]);	//2号叠片	隔膜卷径超声波检测
arrFilter_AD[5].iMode:=2;
arrFilter_AD[5].fPointNum:=20;

arrFilter_AD[6].AD	:=ABS(AI40[2]);	//2号叠片	隔膜放卷纠偏前检测
arrFilter_AD[6].iMode:=2;
arrFilter_AD[6].fPointNum:=20;//30;

arrFilter_AD[7].AD	:=ABS(AI40[3]);	//2号叠片	隔膜放卷纠偏后检测
arrFilter_AD[7].iMode:=2;
arrFilter_AD[7].fPointNum:=20;//30;

//arrFilter_AD[8].AD	:=ABS(AI40[4]);//2号叠片	隔膜张力检测
arrFilter_ADV2[2].AD	:=ABS(AI40[4]);//2号叠片	隔膜张力检测
arrFilter_ADV2[2].iMode:=2;
arrFilter_ADV2[2].fPointNum:=1000;
//3号叠片
arrFilter_AD[9].AD	:=ABS(AI50[1]);	//3号叠片	隔膜卷径超声波检测
arrFilter_AD[9].iMode:=2;
arrFilter_AD[9].fPointNum:=20;

arrFilter_AD[10].AD	:=ABS(AI50[2]);	//3号叠片	隔膜放卷纠偏前检测
arrFilter_AD[10].iMode:=2;
arrFilter_AD[10].fPointNum:=20;//30;

arrFilter_AD[11].AD	:=ABS(AI50[3]);	//3号叠片	隔膜放卷纠偏后检测
arrFilter_AD[11].iMode:=2;
arrFilter_AD[11].fPointNum:=20;//30;

//arrFilter_AD[12].AD	:=ABS(AI50[4]);//3号叠片	隔膜张力检测
arrFilter_ADV2[3].AD	:=ABS(AI50[4]);//3号叠片	隔膜张力检测
arrFilter_ADV2[3].iMode:=2;
arrFilter_ADV2[3].fPointNum:=1000;

FOR  I1:=1 TO  12  DO//MaxAINo
	IF  I1=4  THEN
           arrFilter_ADV2[1](
			  iMode:=         , 
			  AD:=				arrFilter_ADV2[1].AD, 
			  iLimitH:=         parFilterAD[4].iLimitH  , 
			  iLimitL:=          parFilterAD[4].iLimitL   , 
			  fRangeH:=      parFilterAD[4].fRangeH , 
			  fRangeL:=       parFilterAD[4].fRangeL , 
			  fPointNum:=    , 
			  Out_Value=>    );
  ELSIF  I1=8 THEN
           arrFilter_ADV2[2](
			  iMode:=         , 
			  AD:=			    arrFilter_ADV2[2].AD, 
			  iLimitH:=         parFilterAD[8].iLimitH  , 
			  iLimitL:=          parFilterAD[8].iLimitL   , 
			  fRangeH:=      parFilterAD[8].fRangeH , 
			  fRangeL:=       parFilterAD[8].fRangeL , 
			  fPointNum:=    , 
			  Out_Value=>);
  ELSIF  I1=12 THEN
           arrFilter_ADV2[3](
			  iMode:=         , 
			  AD:=				arrFilter_ADV2[3].AD, 
			  iLimitH:=         parFilterAD[12].iLimitH  , 
			  iLimitL:=          parFilterAD[12].iLimitL   , 
			  fRangeH:=      parFilterAD[12].fRangeH , 
			  fRangeL:=       parFilterAD[12].fRangeL , 
			  fPointNum:=    , 
			  Out_Value=>);
ELSE
	  arrFilter_AD[I1](
		  iMode:=         , 
		  AD:=				arrFilter_AD[I1].AD               , 
		  iLimitH:=         parFilterAD[I1].iLimitH  , 
		  iLimitL:=          parFilterAD[I1].iLimitL   , 
		  fRangeH:=      parFilterAD[I1].fRangeH , 
		  fRangeL:=       parFilterAD[I1].fRangeL , 
		  fPointNum:=    , 
		  Out_Value=>);
END_IF

END_FOR
//一号叠台
//P2M1_MachCtrl.DT_b.fWindDiameter:=arrFilter_AD[1].Out_Value;
P2M1_MachCtrl.DT_b.RecDevPV:=arrFilter_AD[2].Out_Value;
P2M1_MachCtrl.DT_b.RecDevPV1:=arrFilter_AD[3].Out_Value;
P2M1_MachCtrl.DT_b.TenAnglePos:=LREAL_TO_REAL(arrAxis[P2M1_Axise.AxisName.SEPTATension].NcToPlc.ActPos);	
P2M1_Par.stDT_date.fRectifyMaxValue:= parFilterAD[2].fRangeH;
P2M1_Par.stDT_date.fRectifyMinValue:=parFilterAD[2].fRangeL;
arrFilter_ADV2[1].Out_Value;

//二号叠台
//P2M2_MachCtrl.DT_b.fWindDiameter:=arrFilter_AD[5].Out_Value;
P2M2_MachCtrl.DT_b.RecDevPV:=arrFilter_AD[6].Out_Value;
P2M2_MachCtrl.DT_b.RecDevPV1:=arrFilter_AD[7].Out_Value;
P2M2_MachCtrl.DT_b.TenAnglePos:=LREAL_TO_REAL(arrAxis[P2M2_Axise.AxisName.SEPTATension].NcToPlc.ActPos);	//2号叠片	隔膜张力检测;
P2M2_Par.stDT_date.fRectifyMaxValue:= parFilterAD[6].fRangeH;
P2M2_Par.stDT_date.fRectifyMinValue:=parFilterAD[6].fRangeL;
arrFilter_ADV2[2].Out_Value;
//三号叠台
//P2M3_MachCtrl.DT_b.fWindDiameter:=arrFilter_AD[9].Out_Value;
P2M3_MachCtrl.DT_b.RecDevPV:=arrFilter_AD[10].Out_Value;
P2M3_MachCtrl.DT_b.RecDevPV1:=arrFilter_AD[11].Out_Value;
P2M3_MachCtrl.DT_b.TenAnglePos:=LREAL_TO_REAL(arrAxis[P2M3_Axise.AxisName.SEPTATension].NcToPlc.ActPos);	//3号叠片	隔膜张力检测
P2M3_Par.stDT_date.fRectifyMaxValue:= parFilterAD[10].fRangeH;
P2M3_Par.stDT_date.fRectifyMinValue:=parFilterAD[10].fRangeL;
arrFilter_ADV2[3].Out_Value;
END_ACTION

ACTION AO:
;
END_ACTION

ACTION LimitSwitch:

//1号叠台
arrAxisCtrl[P2AxisNo.P2M1_AnCarryingLine].Io.DigitalInputs;//一号叠台正极搬运平移//直线电机
arrAxisCtrl[P2AxisNo.P2M1_AnCarryingLine].Io.biPosLimit:= arrAxisCtrl[P2AxisNo.P2M1_AnCarryingLine].Io.DigitalInputs.17;
arrAxisCtrl[P2AxisNo.P2M1_AnCarryingLine].Io.biNegLimit:=  arrAxisCtrl[P2AxisNo.P2M1_AnCarryingLine].Io.DigitalInputs.18;
arrAxisCtrl[P2AxisNo.P2M1_AnCarryingLine].Io.biHomeSwitch:=arrAxisCtrl[P2AxisNo.P2M1_AnCarryingLine].Io.DigitalInputs.20;

arrAxisCtrl[P2AxisNo.P2M1_AnCarryingUpDown].Io.DigitalInputs;//一号叠台正极送片搬运升降
arrAxisCtrl[P2AxisNo.P2M1_AnCarryingUpDown].Io.biPosLimit:= arrAxisCtrl[P2AxisNo.P2M1_AnCarryingUpDown].Io.DigitalInputs.16;
arrAxisCtrl[P2AxisNo.P2M1_AnCarryingUpDown].Io.biNegLimit:=  arrAxisCtrl[P2AxisNo.P2M1_AnCarryingUpDown].Io.DigitalInputs.2;
arrAxisCtrl[P2AxisNo.P2M1_AnCarryingUpDown].Io.biHomeSwitch:=arrAxisCtrl[P2AxisNo.P2M1_AnCarryingUpDown].Io.DigitalInputs.2;

arrAxisCtrl[P2AxisNo.P2M1_AnCarryingWhirling].Io.DigitalInputs;//一号叠台正极搬运旋转
arrAxisCtrl[P2AxisNo.P2M1_AnCarryingWhirling].Io.biPosLimit:= arrAxisCtrl[P2AxisNo.P2M1_AnCarryingWhirling].Io.DigitalInputs.16;
arrAxisCtrl[P2AxisNo.P2M1_AnCarryingWhirling].Io.biNegLimit:=  arrAxisCtrl[P2AxisNo.P2M1_AnCarryingWhirling].Io.DigitalInputs.2;
arrAxisCtrl[P2AxisNo.P2M1_AnCarryingWhirling].Io.biHomeSwitch:=arrAxisCtrl[P2AxisNo.P2M1_AnCarryingWhirling].Io.DigitalInputs.2;

arrAxisCtrl[P2AxisNo.P2M1_AndeviationX1].Io.DigitalInputs;//一号叠台正极纠偏平台X1
arrAxisCtrl[P2AxisNo.P2M1_AndeviationX1].Io.biPosLimit:= arrAxisCtrl[P2AxisNo.P2M1_AndeviationX1].Io.DigitalInputs.16;
arrAxisCtrl[P2AxisNo.P2M1_AndeviationX1].Io.biNegLimit:=  arrAxisCtrl[P2AxisNo.P2M1_AndeviationX1].Io.DigitalInputs.17;
arrAxisCtrl[P2AxisNo.P2M1_AndeviationX1].Io.biHomeSwitch:=arrAxisCtrl[P2AxisNo.P2M1_AndeviationX1].Io.DigitalInputs.2;

arrAxisCtrl[P2AxisNo.P2M1_AndeviationX2].Io.DigitalInputs;//一号叠台正极纠偏平台X2
arrAxisCtrl[P2AxisNo.P2M1_AndeviationX2].Io.biPosLimit:= arrAxisCtrl[P2AxisNo.P2M1_AndeviationX2].Io.DigitalInputs.16;
arrAxisCtrl[P2AxisNo.P2M1_AndeviationX2].Io.biNegLimit:=  arrAxisCtrl[P2AxisNo.P2M1_AndeviationX2].Io.DigitalInputs.17;
arrAxisCtrl[P2AxisNo.P2M1_AndeviationX2].Io.biHomeSwitch:=arrAxisCtrl[P2AxisNo.P2M1_AndeviationX2].Io.DigitalInputs.2;

arrAxisCtrl[P2AxisNo.P2M1_AndeviationY].Io.DigitalInputs;//一号叠台正极纠偏平台Y
arrAxisCtrl[P2AxisNo.P2M1_AndeviationY].Io.biPosLimit:= arrAxisCtrl[P2AxisNo.P2M1_AndeviationY].Io.DigitalInputs.16;
arrAxisCtrl[P2AxisNo.P2M1_AndeviationY].Io.biNegLimit:=  arrAxisCtrl[P2AxisNo.P2M1_AndeviationY].Io.DigitalInputs.17;
arrAxisCtrl[P2AxisNo.P2M1_AndeviationY].Io.biHomeSwitch:=arrAxisCtrl[P2AxisNo.P2M1_AndeviationY].Io.DigitalInputs.2;

arrAxisCtrl[P2AxisNo.P2M1_AnDTCarryingLine].Io.DigitalInputs;//一号叠台正极搬运平移1//直线电机
arrAxisCtrl[P2AxisNo.P2M1_AnDTCarryingLine].Io.biPosLimit:=  arrAxisCtrl[P2AxisNo.P2M1_AnDTCarryingLine].Io.DigitalInputs.17;
arrAxisCtrl[P2AxisNo.P2M1_AnDTCarryingLine].Io.biNegLimit:=   arrAxisCtrl[P2AxisNo.P2M1_AnDTCarryingLine].Io.DigitalInputs.18;
arrAxisCtrl[P2AxisNo.P2M1_AnDTCarryingLine].Io.biHomeSwitch:=arrAxisCtrl[P2AxisNo.P2M1_AnDTCarryingLine].Io.DigitalInputs.20;

arrAxisCtrl[P2AxisNo.P2M1_AnDTCarryingUpDown].Io.DigitalInputs;//一号叠台正极搬运升降
arrAxisCtrl[P2AxisNo.P2M1_AnDTCarryingUpDown].Io.biPosLimit:= arrAxisCtrl[P2AxisNo.P2M1_AnDTCarryingUpDown].Io.DigitalInputs.16;
arrAxisCtrl[P2AxisNo.P2M1_AnDTCarryingUpDown].Io.biNegLimit:=  arrAxisCtrl[P2AxisNo.P2M1_AnDTCarryingUpDown].Io.DigitalInputs.2;
arrAxisCtrl[P2AxisNo.P2M1_AnDTCarryingUpDown].Io.biHomeSwitch:=arrAxisCtrl[P2AxisNo.P2M1_AnDTCarryingUpDown].Io.DigitalInputs.2;

arrAxisCtrl[P2AxisNo.P2M1_CaBelt].Io.DigitalInputs;//一号叠台正极送片皮带
//arrAxisCtrl[P2AxisNo.P2M1_CaBelt].Io.biPosLimit:= arrAxisCtrl[P2AxisNo.P2M1_CaBelt].Io.DigitalInputs.16;
//arrAxisCtrl[P2AxisNo.P2M1_CaBelt].Io.biNegLimit:=  arrAxisCtrl[P2AxisNo.P2M1_CaBelt].Io.DigitalInputs.17;
//arrAxisCtrl[P2AxisNo.P2M1_CaBelt].Io.biHomeSwitch:=arrAxisCtrl[P2AxisNo.P2M1_CaBelt].Io.DigitalInputs.2;

arrAxisCtrl[P2AxisNo.P2M1_CaCarryingLine1].Io.DigitalInputs;//一号叠台负极搬运平移1//直线电机
arrAxisCtrl[P2AxisNo.P2M1_CaCarryingLine1].Io.biPosLimit:=  arrAxisCtrl[P2AxisNo.P2M1_CaCarryingLine1].Io.DigitalInputs.17;
arrAxisCtrl[P2AxisNo.P2M1_CaCarryingLine1].Io.biNegLimit:=  arrAxisCtrl[P2AxisNo.P2M1_CaCarryingLine1].Io.DigitalInputs.18;
arrAxisCtrl[P2AxisNo.P2M1_CaCarryingLine1].Io.biHomeSwitch:=arrAxisCtrl[P2AxisNo.P2M1_CaCarryingLine1].Io.DigitalInputs.20;

arrAxisCtrl[P2AxisNo.P2M1_CaCarryingLine2].Io.DigitalInputs;//一号叠台负极搬运平移2//直线电机
arrAxisCtrl[P2AxisNo.P2M1_CaCarryingLine2].Io.biPosLimit:= arrAxisCtrl[P2AxisNo.P2M1_CaCarryingLine2].Io.DigitalInputs.17;
arrAxisCtrl[P2AxisNo.P2M1_CaCarryingLine2].Io.biNegLimit:=  arrAxisCtrl[P2AxisNo.P2M1_CaCarryingLine2].Io.DigitalInputs.18;
arrAxisCtrl[P2AxisNo.P2M1_CaCarryingLine2].Io.biHomeSwitch:=arrAxisCtrl[P2AxisNo.P2M1_CaCarryingLine2].Io.DigitalInputs.20;

arrAxisCtrl[P2AxisNo.P2M1_CaCarryingUpDown1].Io.DigitalInputs;//一号叠台负极送片搬运1升降
arrAxisCtrl[P2AxisNo.P2M1_CaCarryingUpDown1].Io.biPosLimit:= arrAxisCtrl[P2AxisNo.P2M1_CaCarryingUpDown1].Io.DigitalInputs.16;
arrAxisCtrl[P2AxisNo.P2M1_CaCarryingUpDown1].Io.biNegLimit:=  arrAxisCtrl[P2AxisNo.P2M1_CaCarryingUpDown1].Io.DigitalInputs.2;
arrAxisCtrl[P2AxisNo.P2M1_CaCarryingUpDown1].Io.biHomeSwitch:=arrAxisCtrl[P2AxisNo.P2M1_CaCarryingUpDown1].Io.DigitalInputs.2;

arrAxisCtrl[P2AxisNo.P2M1_CaCarryingUpDown2].Io.DigitalInputs;//一号叠台负极送片搬运2升降
arrAxisCtrl[P2AxisNo.P2M1_CaCarryingUpDown2].Io.biPosLimit:= arrAxisCtrl[P2AxisNo.P2M1_CaCarryingUpDown2].Io.DigitalInputs.16;
arrAxisCtrl[P2AxisNo.P2M1_CaCarryingUpDown2].Io.biNegLimit:=  arrAxisCtrl[P2AxisNo.P2M1_CaCarryingUpDown2].Io.DigitalInputs.2;
arrAxisCtrl[P2AxisNo.P2M1_CaCarryingUpDown2].Io.biHomeSwitch:=arrAxisCtrl[P2AxisNo.P2M1_CaCarryingUpDown2].Io.DigitalInputs.2;

arrAxisCtrl[P2AxisNo.P2M1_CaCarryingWhirling1].Io.DigitalInputs;//一号叠台负极送片搬运1旋转
arrAxisCtrl[P2AxisNo.P2M1_CaCarryingWhirling1].Io.biPosLimit:= arrAxisCtrl[P2AxisNo.P2M1_CaCarryingWhirling1].Io.DigitalInputs.16;
arrAxisCtrl[P2AxisNo.P2M1_CaCarryingWhirling1].Io.biNegLimit:=  arrAxisCtrl[P2AxisNo.P2M1_CaCarryingWhirling1].Io.DigitalInputs.2;
arrAxisCtrl[P2AxisNo.P2M1_CaCarryingWhirling1].Io.biHomeSwitch:=arrAxisCtrl[P2AxisNo.P2M1_CaCarryingWhirling1].Io.DigitalInputs.2;

arrAxisCtrl[P2AxisNo.P2M1_CadeviationX1].Io.DigitalInputs;//一号叠台负极纠偏平台X1
arrAxisCtrl[P2AxisNo.P2M1_CadeviationX1].Io.biPosLimit:= arrAxisCtrl[P2AxisNo.P2M1_CadeviationX1].Io.DigitalInputs.16;
arrAxisCtrl[P2AxisNo.P2M1_CadeviationX1].Io.biNegLimit:=  arrAxisCtrl[P2AxisNo.P2M1_CadeviationX1].Io.DigitalInputs.17;
arrAxisCtrl[P2AxisNo.P2M1_CadeviationX1].Io.biHomeSwitch:=arrAxisCtrl[P2AxisNo.P2M1_CadeviationX1].Io.DigitalInputs.2;

arrAxisCtrl[P2AxisNo.P2M1_CadeviationX2].Io.DigitalInputs;//一号叠台负极纠偏平台X2
arrAxisCtrl[P2AxisNo.P2M1_CadeviationX2].Io.biPosLimit:= arrAxisCtrl[P2AxisNo.P2M1_CadeviationX2].Io.DigitalInputs.16;
arrAxisCtrl[P2AxisNo.P2M1_CadeviationX2].Io.biNegLimit:=  arrAxisCtrl[P2AxisNo.P2M1_CadeviationX2].Io.DigitalInputs.17;
arrAxisCtrl[P2AxisNo.P2M1_CadeviationX2].Io.biHomeSwitch:=arrAxisCtrl[P2AxisNo.P2M1_CadeviationX2].Io.DigitalInputs.2;

arrAxisCtrl[P2AxisNo.P2M1_CadeviationY].Io.DigitalInputs;//一号叠台负极纠偏平台Y
arrAxisCtrl[P2AxisNo.P2M1_CadeviationY].Io.biPosLimit:= arrAxisCtrl[P2AxisNo.P2M1_CadeviationY].Io.DigitalInputs.16;
arrAxisCtrl[P2AxisNo.P2M1_CadeviationY].Io.biNegLimit:=  arrAxisCtrl[P2AxisNo.P2M1_CadeviationY].Io.DigitalInputs.17;
arrAxisCtrl[P2AxisNo.P2M1_CadeviationY].Io.biHomeSwitch:=arrAxisCtrl[P2AxisNo.P2M1_CadeviationY].Io.DigitalInputs.2;

arrAxisCtrl[P2AxisNo.P2M1_CaDTCarryingLine].Io.DigitalInputs;//一号叠台负极搬运平移//直线电机
arrAxisCtrl[P2AxisNo.P2M1_CaDTCarryingLine].Io.biPosLimit:= arrAxisCtrl[P2AxisNo.P2M1_CaDTCarryingLine].Io.DigitalInputs.17;
arrAxisCtrl[P2AxisNo.P2M1_CaDTCarryingLine].Io.biNegLimit:=  arrAxisCtrl[P2AxisNo.P2M1_CaDTCarryingLine].Io.DigitalInputs.18;
arrAxisCtrl[P2AxisNo.P2M1_CaDTCarryingLine].Io.biHomeSwitch:=arrAxisCtrl[P2AxisNo.P2M1_CaDTCarryingLine].Io.DigitalInputs.20;

arrAxisCtrl[P2AxisNo.P2M1_CaDTCarryingUpDown].Io.DigitalInputs;//一号叠台负极叠片搬运升降
arrAxisCtrl[P2AxisNo.P2M1_CaDTCarryingUpDown].Io.biPosLimit:= arrAxisCtrl[P2AxisNo.P2M1_CaDTCarryingUpDown].Io.DigitalInputs.16;
arrAxisCtrl[P2AxisNo.P2M1_CaDTCarryingUpDown].Io.biNegLimit:=  arrAxisCtrl[P2AxisNo.P2M1_CaDTCarryingUpDown].Io.DigitalInputs.2;
arrAxisCtrl[P2AxisNo.P2M1_CaDTCarryingUpDown].Io.biHomeSwitch:=arrAxisCtrl[P2AxisNo.P2M1_CaDTCarryingUpDown].Io.DigitalInputs.2;

arrAxisCtrl[P2AxisNo.P2M1_DTUpDown].Io.DigitalInputs;//一号叠台升降
arrAxisCtrl[P2AxisNo.P2M1_DTUpDown].Io.biPosLimit:= arrAxisCtrl[P2AxisNo.P2M1_DTUpDown].Io.DigitalInputs.16;
arrAxisCtrl[P2AxisNo.P2M1_DTUpDown].Io.biNegLimit:=  arrAxisCtrl[P2AxisNo.P2M1_DTUpDown].Io.DigitalInputs.2;
arrAxisCtrl[P2AxisNo.P2M1_DTUpDown].Io.biHomeSwitch:=arrAxisCtrl[P2AxisNo.P2M1_DTUpDown].Io.DigitalInputs.2;


////////////////////////////////////
arrAxisCtrl[P2AxisNo.P2M1_GluingLine].Io.DigitalInputs;//一号叠台侧胶夹平移
arrAxisCtrl[P2AxisNo.P2M1_GluingLine].Io.biPosLimit:= arrAxisCtrl[P2AxisNo.P2M1_GluingLine].Io.DigitalInputs.16;
arrAxisCtrl[P2AxisNo.P2M1_GluingLine].Io.biNegLimit:=  arrAxisCtrl[P2AxisNo.P2M1_GluingLine].Io.DigitalInputs.17;
arrAxisCtrl[P2AxisNo.P2M1_GluingLine].Io.biHomeSwitch:=arrAxisCtrl[P2AxisNo.P2M1_GluingLine].Io.DigitalInputs.2;

arrAxisCtrl[P2AxisNo.P2M1_GluingRetracting].Io.DigitalInputs;//一号叠台贴胶头进退
arrAxisCtrl[P2AxisNo.P2M1_GluingRetracting].Io.biPosLimit:= arrAxisCtrl[P2AxisNo.P2M1_GluingRetracting].Io.DigitalInputs.16;
arrAxisCtrl[P2AxisNo.P2M1_GluingRetracting].Io.biNegLimit:=  arrAxisCtrl[P2AxisNo.P2M1_GluingRetracting].Io.DigitalInputs.17;
arrAxisCtrl[P2AxisNo.P2M1_GluingRetracting].Io.biHomeSwitch:=arrAxisCtrl[P2AxisNo.P2M1_GluingRetracting].Io.DigitalInputs.2;

arrAxisCtrl[P2AxisNo.P2M1_GluingUpDown].Io.DigitalInputs;//一号叠台拉胶升降
arrAxisCtrl[P2AxisNo.P2M1_GluingUpDown].Io.biPosLimit:= arrAxisCtrl[P2AxisNo.P2M1_GluingUpDown].Io.DigitalInputs.16;
arrAxisCtrl[P2AxisNo.P2M1_GluingUpDown].Io.biNegLimit:=  arrAxisCtrl[P2AxisNo.P2M1_GluingUpDown].Io.DigitalInputs.17;
arrAxisCtrl[P2AxisNo.P2M1_GluingUpDown].Io.biHomeSwitch:=arrAxisCtrl[P2AxisNo.P2M1_GluingUpDown].Io.DigitalInputs.2;

arrAxisCtrl[P2AxisNo.P2M1_GluingWhirling].Io.DigitalInputs;//一号叠台侧胶夹旋转
arrAxisCtrl[P2AxisNo.P2M1_GluingWhirling].Io.biPosLimit:= arrAxisCtrl[P2AxisNo.P2M1_GluingWhirling].Io.DigitalInputs.16;
arrAxisCtrl[P2AxisNo.P2M1_GluingWhirling].Io.biNegLimit:=  arrAxisCtrl[P2AxisNo.P2M1_GluingWhirling].Io.DigitalInputs.17;
arrAxisCtrl[P2AxisNo.P2M1_GluingWhirling].Io.biHomeSwitch:=arrAxisCtrl[P2AxisNo.P2M1_GluingWhirling].Io.DigitalInputs.2;

arrAxisCtrl[P2AxisNo.P2M1_LCurlingneedleLine].Io.DigitalInputs;//一号叠台长卷针平移   雷赛
arrAxisCtrl[P2AxisNo.P2M1_LCurlingneedleLine].Io.biPosLimit:= arrAxisCtrl[P2AxisNo.P2M1_LCurlingneedleLine].Io.DigitalInputs.6;
arrAxisCtrl[P2AxisNo.P2M1_LCurlingneedleLine].Io.biNegLimit:=  arrAxisCtrl[P2AxisNo.P2M1_LCurlingneedleLine].Io.DigitalInputs.7;
arrAxisCtrl[P2AxisNo.P2M1_LCurlingneedleLine].Io.biHomeSwitch:=arrAxisCtrl[P2AxisNo.P2M1_LCurlingneedleLine].Io.DigitalInputs.7;

arrAxisCtrl[P2AxisNo.P2M1_LCurlingneedleWhirling].Io.DigitalInputs;//一号叠台长卷针旋转  雷赛
//arrAxisCtrl[P2AxisNo.P2M1_LCurlingneedleWhirling].Io.biPosLimit:= arrAxisCtrl[P2AxisNo.P2M1_LCurlingneedleWhirling].Io.DigitalInputs.6;
//arrAxisCtrl[P2AxisNo.P2M1_LCurlingneedleWhirling].Io.biNegLimit:=  arrAxisCtrl[P2AxisNo.P2M1_LCurlingneedleWhirling].Io.DigitalInputs.7;
arrAxisCtrl[P2AxisNo.P2M1_LCurlingneedleWhirling].Io.biHomeSwitch:=arrAxisCtrl[P2AxisNo.P2M1_LCurlingneedleWhirling].Io.DigitalInputs.2;




/////////////////
arrAxisCtrl[P2AxisNo.P2M1_LeftYDLine].Io.DigitalInputs;//一号叠台左压刀开合
arrAxisCtrl[P2AxisNo.P2M1_LeftYDLine].Io.biPosLimit:= arrAxisCtrl[P2AxisNo.P2M1_LeftYDLine].Io.DigitalInputs.16;
arrAxisCtrl[P2AxisNo.P2M1_LeftYDLine].Io.biNegLimit:=  arrAxisCtrl[P2AxisNo.P2M1_LeftYDLine].Io.DigitalInputs.2;
arrAxisCtrl[P2AxisNo.P2M1_LeftYDLine].Io.biHomeSwitch:=arrAxisCtrl[P2AxisNo.P2M1_LeftYDLine].Io.DigitalInputs.2;

arrAxisCtrl[P2AxisNo.P2M1_LeftYDUpDown].Io.DigitalInputs;//一号叠台左压刀升降
arrAxisCtrl[P2AxisNo.P2M1_LeftYDUpDown].Io.biPosLimit:= arrAxisCtrl[P2AxisNo.P2M1_LeftYDUpDown].Io.DigitalInputs.16;
arrAxisCtrl[P2AxisNo.P2M1_LeftYDUpDown].Io.biNegLimit:=  arrAxisCtrl[P2AxisNo.P2M1_LeftYDUpDown].Io.DigitalInputs.2;
arrAxisCtrl[P2AxisNo.P2M1_LeftYDUpDown].Io.biHomeSwitch:=arrAxisCtrl[P2AxisNo.P2M1_LeftYDUpDown].Io.DigitalInputs.2;

arrAxisCtrl[P2AxisNo.P2M1_RightYDLine].Io.DigitalInputs;//一号叠台右压刀开合
arrAxisCtrl[P2AxisNo.P2M1_RightYDLine].Io.biPosLimit:= arrAxisCtrl[P2AxisNo.P2M1_RightYDLine].Io.DigitalInputs.16;
arrAxisCtrl[P2AxisNo.P2M1_RightYDLine].Io.biNegLimit:=  arrAxisCtrl[P2AxisNo.P2M1_RightYDLine].Io.DigitalInputs.2;
arrAxisCtrl[P2AxisNo.P2M1_RightYDLine].Io.biHomeSwitch:=arrAxisCtrl[P2AxisNo.P2M1_RightYDLine].Io.DigitalInputs.2;

arrAxisCtrl[P2AxisNo.P2M1_RightYDUpDown].Io.DigitalInputs;//右压刀升降
arrAxisCtrl[P2AxisNo.P2M1_RightYDUpDown].Io.biPosLimit:= arrAxisCtrl[P2AxisNo.P2M1_RightYDUpDown].Io.DigitalInputs.16;
arrAxisCtrl[P2AxisNo.P2M1_RightYDUpDown].Io.biNegLimit:=  arrAxisCtrl[P2AxisNo.P2M1_RightYDUpDown].Io.DigitalInputs.2;
arrAxisCtrl[P2AxisNo.P2M1_RightYDUpDown].Io.biHomeSwitch:=arrAxisCtrl[P2AxisNo.P2M1_RightYDUpDown].Io.DigitalInputs.2;


////////////////
arrAxisCtrl[P2AxisNo.P2M1_SCurlingneedleLine].Io.DigitalInputs;//一号叠台平卷针平移   雷赛
arrAxisCtrl[P2AxisNo.P2M1_SCurlingneedleLine].Io.biPosLimit:= arrAxisCtrl[P2AxisNo.P2M1_SCurlingneedleLine].Io.DigitalInputs.6;
arrAxisCtrl[P2AxisNo.P2M1_SCurlingneedleLine].Io.biNegLimit:=  arrAxisCtrl[P2AxisNo.P2M1_SCurlingneedleLine].Io.DigitalInputs.7;
arrAxisCtrl[P2AxisNo.P2M1_SCurlingneedleLine].Io.biHomeSwitch:=arrAxisCtrl[P2AxisNo.P2M1_SCurlingneedleLine].Io.DigitalInputs.7;

arrAxisCtrl[P2AxisNo.P2M1_SCurlingneedleWhirling].Io.DigitalInputs;//一号叠台短卷针旋转   雷赛
//arrAxisCtrl[P2AxisNo.P2M1_SCurlingneedleWhirling].Io.biPosLimit:= arrAxisCtrl[P2AxisNo.P2M1_SCurlingneedleWhirling].Io.DigitalInputs.6;
//arrAxisCtrl[P2AxisNo.P2M1_SCurlingneedleWhirling].Io.biNegLimit:=  arrAxisCtrl[P2AxisNo.P2M1_SCurlingneedleWhirling].Io.DigitalInputs.7;
arrAxisCtrl[P2AxisNo.P2M1_SCurlingneedleWhirling].Io.biHomeSwitch:=arrAxisCtrl[P2AxisNo.P2M1_SCurlingneedleWhirling].Io.DigitalInputs.2;



arrAxisCtrl[P2AxisNo.P2M1_SEPTAdeviation1].Io.DigitalInputs;//一号叠台隔膜放卷纠偏
arrAxisCtrl[P2AxisNo.P2M1_SEPTAdeviation1].Io.biPosLimit:= arrAxisCtrl[P2AxisNo.P2M1_SEPTAdeviation1].Io.DigitalInputs.16;
arrAxisCtrl[P2AxisNo.P2M1_SEPTAdeviation1].Io.biNegLimit:=  arrAxisCtrl[P2AxisNo.P2M1_SEPTAdeviation1].Io.DigitalInputs.2;
arrAxisCtrl[P2AxisNo.P2M1_SEPTAdeviation1].Io.biHomeSwitch:=arrAxisCtrl[P2AxisNo.P2M1_SEPTAdeviation1].Io.DigitalInputs.2;

arrAxisCtrl[P2AxisNo.P2M1_SEPTAdeviation2].Io.DigitalInputs;//一号叠台隔膜尾部纠偏
arrAxisCtrl[P2AxisNo.P2M1_SEPTAdeviation2].Io.biPosLimit:= arrAxisCtrl[P2AxisNo.P2M1_SEPTAdeviation2].Io.DigitalInputs.16;
arrAxisCtrl[P2AxisNo.P2M1_SEPTAdeviation2].Io.biNegLimit:=  arrAxisCtrl[P2AxisNo.P2M1_SEPTAdeviation2].Io.DigitalInputs.2;
arrAxisCtrl[P2AxisNo.P2M1_SEPTAdeviation2].Io.biHomeSwitch:=arrAxisCtrl[P2AxisNo.P2M1_SEPTAdeviation2].Io.DigitalInputs.2;

arrAxisCtrl[P2AxisNo.P2M1_SEPTATCache].Io.DigitalInputs;//一号叠台隔膜缓存//直线电机
arrAxisCtrl[P2AxisNo.P2M1_SEPTATCache].Io.biPosLimit:= arrAxisCtrl[P2AxisNo.P2M1_SEPTATCache].Io.DigitalInputs.17;
arrAxisCtrl[P2AxisNo.P2M1_SEPTATCache].Io.biNegLimit:=  arrAxisCtrl[P2AxisNo.P2M1_SEPTATCache].Io.DigitalInputs.18;
arrAxisCtrl[P2AxisNo.P2M1_SEPTATCache].Io.biHomeSwitch:=arrAxisCtrl[P2AxisNo.P2M1_SEPTATCache].Io.DigitalInputs.20;

arrAxisCtrl[P2AxisNo.P2M1_SEPTATension].Io.DigitalInputs;//一号叠台隔膜摆杆张力
//arrAxisCtrl[P2AxisNo.P2M1_SEPTATension].Io.biPosLimit:= arrAxisCtrl[P2AxisNo.P2M1_SEPTATension].Io.DigitalInputs.16;
//arrAxisCtrl[P2AxisNo.P2M1_SEPTATension].Io.biNegLimit:=  arrAxisCtrl[P2AxisNo.P2M1_SEPTATension].Io.DigitalInputs.17;
//arrAxisCtrl[P2AxisNo.P2M1_SEPTATension].Io.biHomeSwitch:=arrAxisCtrl[P2AxisNo.P2M1_SEPTATension].Io.DigitalInputs.2;

arrAxisCtrl[P2AxisNo.P2M1_SEPTATLine].Io.DigitalInputs;//一号叠台隔膜平移//直线电机
arrAxisCtrl[P2AxisNo.P2M1_SEPTATLine].Io.biPosLimit:= arrAxisCtrl[P2AxisNo.P2M1_SEPTATLine].Io.DigitalInputs.17;
arrAxisCtrl[P2AxisNo.P2M1_SEPTATLine].Io.biNegLimit:=  arrAxisCtrl[P2AxisNo.P2M1_SEPTATLine].Io.DigitalInputs.18;
arrAxisCtrl[P2AxisNo.P2M1_SEPTATLine].Io.biHomeSwitch:=arrAxisCtrl[P2AxisNo.P2M1_SEPTATLine].Io.DigitalInputs.20;

arrAxisCtrl[P2AxisNo.P2M1_SEPTAunwinding].Io.DigitalInputs;//一号叠台隔膜放卷
//arrAxisCtrl[P2AxisNo.P2M1_SEPTAunwinding].Io.biPosLimit:= arrAxisCtrl[P2AxisNo.P2M1_SEPTAunwinding].Io.DigitalInputs.16;
//arrAxisCtrl[P2AxisNo.P2M1_SEPTAunwinding].Io.biNegLimit:=  arrAxisCtrl[P2AxisNo.P2M1_SEPTAunwinding].Io.DigitalInputs.17;
//arrAxisCtrl[P2AxisNo.P2M1_SEPTAunwinding].Io.biHomeSwitch:=arrAxisCtrl[P2AxisNo.P2M1_SEPTAunwinding].Io.DigitalInputs.2;

arrAxisCtrl[P2AxisNo.P2M1_TailCurlLine].Io.DigitalInputs;//一号叠台尾卷夹电芯平移
arrAxisCtrl[P2AxisNo.P2M1_TailCurlLine].Io.biPosLimit:= arrAxisCtrl[P2AxisNo.P2M1_TailCurlLine].Io.DigitalInputs.16;
arrAxisCtrl[P2AxisNo.P2M1_TailCurlLine].Io.biNegLimit:=  arrAxisCtrl[P2AxisNo.P2M1_TailCurlLine].Io.DigitalInputs.17;
arrAxisCtrl[P2AxisNo.P2M1_TailCurlLine].Io.biHomeSwitch:=arrAxisCtrl[P2AxisNo.P2M1_TailCurlLine].Io.DigitalInputs.2;

arrAxisCtrl[P2AxisNo.P2M1_TailCurlRetracting].Io.DigitalInputs;//一号叠台尾卷夹电芯伸缩
arrAxisCtrl[P2AxisNo.P2M1_TailCurlRetracting].Io.biPosLimit:= arrAxisCtrl[P2AxisNo.P2M1_TailCurlRetracting].Io.DigitalInputs.16;
arrAxisCtrl[P2AxisNo.P2M1_TailCurlRetracting].Io.biNegLimit:=  arrAxisCtrl[P2AxisNo.P2M1_TailCurlRetracting].Io.DigitalInputs.2;
arrAxisCtrl[P2AxisNo.P2M1_TailCurlRetracting].Io.biHomeSwitch:=arrAxisCtrl[P2AxisNo.P2M1_TailCurlRetracting].Io.DigitalInputs.2;

arrAxisCtrl[P2AxisNo.P2M1_TailCurlSEPTALine].Io.DigitalInputs;//一号叠台夹膜平移
arrAxisCtrl[P2AxisNo.P2M1_TailCurlSEPTALine].Io.biPosLimit:= arrAxisCtrl[P2AxisNo.P2M1_TailCurlSEPTALine].Io.DigitalInputs.16;
arrAxisCtrl[P2AxisNo.P2M1_TailCurlSEPTALine].Io.biNegLimit:=  arrAxisCtrl[P2AxisNo.P2M1_TailCurlSEPTALine].Io.DigitalInputs.17;
arrAxisCtrl[P2AxisNo.P2M1_TailCurlSEPTALine].Io.biHomeSwitch:=arrAxisCtrl[P2AxisNo.P2M1_TailCurlSEPTALine].Io.DigitalInputs.17;

arrAxisCtrl[P2AxisNo.P2M1_TailCurlSEPTAUpDown].Io.DigitalInputs;//一号叠台夹膜升降
arrAxisCtrl[P2AxisNo.P2M1_TailCurlSEPTAUpDown].Io.biPosLimit:= arrAxisCtrl[P2AxisNo.P2M1_TailCurlSEPTAUpDown].Io.DigitalInputs.16;
arrAxisCtrl[P2AxisNo.P2M1_TailCurlSEPTAUpDown].Io.biNegLimit:=  arrAxisCtrl[P2AxisNo.P2M1_TailCurlSEPTAUpDown].Io.DigitalInputs.2;
arrAxisCtrl[P2AxisNo.P2M1_TailCurlSEPTAUpDown].Io.biHomeSwitch:=arrAxisCtrl[P2AxisNo.P2M1_TailCurlSEPTAUpDown].Io.DigitalInputs.2;

arrAxisCtrl[P2AxisNo.P2M1_TailCurlUpDown].Io.DigitalInputs;//一号叠台尾卷夹电芯升降
arrAxisCtrl[P2AxisNo.P2M1_TailCurlUpDown].Io.biPosLimit:= arrAxisCtrl[P2AxisNo.P2M1_TailCurlUpDown].Io.DigitalInputs.16;
arrAxisCtrl[P2AxisNo.P2M1_TailCurlUpDown].Io.biNegLimit:=  arrAxisCtrl[P2AxisNo.P2M1_TailCurlUpDown].Io.DigitalInputs.17;
arrAxisCtrl[P2AxisNo.P2M1_TailCurlUpDown].Io.biHomeSwitch:=arrAxisCtrl[P2AxisNo.P2M1_TailCurlUpDown].Io.DigitalInputs.2;

arrAxisCtrl[P2AxisNo.P2M1_TailCurlWhirling].Io.DigitalInputs;//一号叠台尾卷夹电芯旋转
arrAxisCtrl[P2AxisNo.P2M1_TailCurlWhirling].Io.biPosLimit:= arrAxisCtrl[P2AxisNo.P2M1_TailCurlWhirling].Io.DigitalInputs.16;
arrAxisCtrl[P2AxisNo.P2M1_TailCurlWhirling].Io.biNegLimit:=  arrAxisCtrl[P2AxisNo.P2M1_TailCurlWhirling].Io.DigitalInputs.17;
arrAxisCtrl[P2AxisNo.P2M1_TailCurlWhirling].Io.biHomeSwitch:=arrAxisCtrl[P2AxisNo.P2M1_TailCurlWhirling].Io.DigitalInputs.17;


//2号叠台
arrAxisCtrl[P2AxisNo.P2M2_AnCarryingLine].Io.DigitalInputs;//二号叠台正极送片搬运平移//直线电机
arrAxisCtrl[P2AxisNo.P2M2_AnCarryingLine].Io.biPosLimit:= arrAxisCtrl[P2AxisNo.P2M2_AnCarryingLine].Io.DigitalInputs.17;
arrAxisCtrl[P2AxisNo.P2M2_AnCarryingLine].Io.biNegLimit:= arrAxisCtrl[P2AxisNo.P2M2_AnCarryingLine].Io.DigitalInputs.18;
arrAxisCtrl[P2AxisNo.P2M2_AnCarryingLine].Io.biHomeSwitch:=arrAxisCtrl[P2AxisNo.P2M2_AnCarryingLine].Io.DigitalInputs.20;

arrAxisCtrl[P2AxisNo.P2M2_AnCarryingUpDown].Io.DigitalInputs;//二号叠台正极送片搬运升降
arrAxisCtrl[P2AxisNo.P2M2_AnCarryingUpDown].Io.biPosLimit:= arrAxisCtrl[P2AxisNo.P2M2_AnCarryingUpDown].Io.DigitalInputs.16;
arrAxisCtrl[P2AxisNo.P2M2_AnCarryingUpDown].Io.biNegLimit:=  arrAxisCtrl[P2AxisNo.P2M2_AnCarryingUpDown].Io.DigitalInputs.2;
arrAxisCtrl[P2AxisNo.P2M2_AnCarryingUpDown].Io.biHomeSwitch:=arrAxisCtrl[P2AxisNo.P2M2_AnCarryingUpDown].Io.DigitalInputs.2;

arrAxisCtrl[P2AxisNo.P2M2_AnCarryingWhirling].Io.DigitalInputs;//二号叠台正极送片搬运旋转
arrAxisCtrl[P2AxisNo.P2M2_AnCarryingWhirling].Io.biPosLimit:= arrAxisCtrl[P2AxisNo.P2M2_AnCarryingWhirling].Io.DigitalInputs.16;
arrAxisCtrl[P2AxisNo.P2M2_AnCarryingWhirling].Io.biNegLimit:=  arrAxisCtrl[P2AxisNo.P2M2_AnCarryingWhirling].Io.DigitalInputs.2;
arrAxisCtrl[P2AxisNo.P2M2_AnCarryingWhirling].Io.biHomeSwitch:=arrAxisCtrl[P2AxisNo.P2M2_AnCarryingWhirling].Io.DigitalInputs.2;

arrAxisCtrl[P2AxisNo.P2M2_AndeviationX1].Io.DigitalInputs;//二号叠台正极纠偏平台X1
arrAxisCtrl[P2AxisNo.P2M2_AndeviationX1].Io.biPosLimit:= arrAxisCtrl[P2AxisNo.P2M2_AndeviationX1].Io.DigitalInputs.16;
arrAxisCtrl[P2AxisNo.P2M2_AndeviationX1].Io.biNegLimit:=  arrAxisCtrl[P2AxisNo.P2M2_AndeviationX1].Io.DigitalInputs.17;
arrAxisCtrl[P2AxisNo.P2M2_AndeviationX1].Io.biHomeSwitch:=arrAxisCtrl[P2AxisNo.P2M2_AndeviationX1].Io.DigitalInputs.2;

arrAxisCtrl[P2AxisNo.P2M2_AndeviationX2].Io.DigitalInputs;//二号叠台正极纠偏平台X2
arrAxisCtrl[P2AxisNo.P2M2_AndeviationX2].Io.biPosLimit:= arrAxisCtrl[P2AxisNo.P2M2_AndeviationX2].Io.DigitalInputs.16;
arrAxisCtrl[P2AxisNo.P2M2_AndeviationX2].Io.biNegLimit:=  arrAxisCtrl[P2AxisNo.P2M2_AndeviationX2].Io.DigitalInputs.17;
arrAxisCtrl[P2AxisNo.P2M2_AndeviationX2].Io.biHomeSwitch:=arrAxisCtrl[P2AxisNo.P2M2_AndeviationX2].Io.DigitalInputs.2;

arrAxisCtrl[P2AxisNo.P2M2_AndeviationY].Io.DigitalInputs;//二号叠台正极纠偏平台Y
arrAxisCtrl[P2AxisNo.P2M2_AndeviationY].Io.biPosLimit:= arrAxisCtrl[P2AxisNo.P2M2_AndeviationY].Io.DigitalInputs.16;
arrAxisCtrl[P2AxisNo.P2M2_AndeviationY].Io.biNegLimit:=  arrAxisCtrl[P2AxisNo.P2M2_AndeviationY].Io.DigitalInputs.17;
arrAxisCtrl[P2AxisNo.P2M2_AndeviationY].Io.biHomeSwitch:=arrAxisCtrl[P2AxisNo.P2M2_AndeviationY].Io.DigitalInputs.2;

arrAxisCtrl[P2AxisNo.P2M2_AnDTCarryingLine].Io.DigitalInputs;//二号叠台正极叠片搬运平移1//直线电机
arrAxisCtrl[P2AxisNo.P2M2_AnDTCarryingLine].Io.biPosLimit:= arrAxisCtrl[P2AxisNo.P2M2_AnDTCarryingLine].Io.DigitalInputs.17;
arrAxisCtrl[P2AxisNo.P2M2_AnDTCarryingLine].Io.biNegLimit:=  arrAxisCtrl[P2AxisNo.P2M2_AnDTCarryingLine].Io.DigitalInputs.18;
arrAxisCtrl[P2AxisNo.P2M2_AnDTCarryingLine].Io.biHomeSwitch:=arrAxisCtrl[P2AxisNo.P2M2_AnDTCarryingLine].Io.DigitalInputs.20;

arrAxisCtrl[P2AxisNo.P2M2_AnDTCarryingUpDown].Io.DigitalInputs;//二号叠台正极叠台搬运升降
arrAxisCtrl[P2AxisNo.P2M2_AnDTCarryingUpDown].Io.biPosLimit:= arrAxisCtrl[P2AxisNo.P2M2_AnDTCarryingUpDown].Io.DigitalInputs.16;
arrAxisCtrl[P2AxisNo.P2M2_AnDTCarryingUpDown].Io.biNegLimit:=  arrAxisCtrl[P2AxisNo.P2M2_AnDTCarryingUpDown].Io.DigitalInputs.2;
arrAxisCtrl[P2AxisNo.P2M2_AnDTCarryingUpDown].Io.biHomeSwitch:=arrAxisCtrl[P2AxisNo.P2M2_AnDTCarryingUpDown].Io.DigitalInputs.2;

arrAxisCtrl[P2AxisNo.P2M2_CaBelt].Io.DigitalInputs;//二号叠台正极送片皮带
//arrAxisCtrl[P2AxisNo.P2M2_CaBelt].Io.biPosLimit:=NOT arrAxisCtrl[P2AxisNo.P2M2_CaBelt].Io.DigitalInputs.16;
//arrAxisCtrl[P2AxisNo.P2M2_CaBelt].Io.biNegLimit:=NOT  arrAxisCtrl[P2AxisNo.P2M2_CaBelt].Io.DigitalInputs.17;
//arrAxisCtrl[P2AxisNo.P2M2_CaBelt].Io.biHomeSwitch:=arrAxisCtrl[P2AxisNo.P2M2_CaBelt].Io.DigitalInputs.2;

arrAxisCtrl[P2AxisNo.P2M2_CaCarryingLine1].Io.DigitalInputs;//二号叠台负极送片搬运1平移//直线电机
arrAxisCtrl[P2AxisNo.P2M2_CaCarryingLine1].Io.biPosLimit:= arrAxisCtrl[P2AxisNo.P2M2_CaCarryingLine1].Io.DigitalInputs.17;
arrAxisCtrl[P2AxisNo.P2M2_CaCarryingLine1].Io.biNegLimit:=  arrAxisCtrl[P2AxisNo.P2M2_CaCarryingLine1].Io.DigitalInputs.18;
arrAxisCtrl[P2AxisNo.P2M2_CaCarryingLine1].Io.biHomeSwitch:=arrAxisCtrl[P2AxisNo.P2M2_CaCarryingLine1].Io.DigitalInputs.20;

arrAxisCtrl[P2AxisNo.P2M2_CaCarryingLine2].Io.DigitalInputs;//二号叠台负极送片搬运2平移//直线电机
arrAxisCtrl[P2AxisNo.P2M2_CaCarryingLine2].Io.biPosLimit:= arrAxisCtrl[P2AxisNo.P2M2_CaCarryingLine2].Io.DigitalInputs.17;
arrAxisCtrl[P2AxisNo.P2M2_CaCarryingLine2].Io.biNegLimit:=  arrAxisCtrl[P2AxisNo.P2M2_CaCarryingLine2].Io.DigitalInputs.18;
arrAxisCtrl[P2AxisNo.P2M2_CaCarryingLine2].Io.biHomeSwitch:=arrAxisCtrl[P2AxisNo.P2M2_CaCarryingLine2].Io.DigitalInputs.20;

arrAxisCtrl[P2AxisNo.P2M2_CaCarryingUpDown1].Io.DigitalInputs;//二号叠台负极送片搬运1升降
arrAxisCtrl[P2AxisNo.P2M2_CaCarryingUpDown1].Io.biPosLimit:= arrAxisCtrl[P2AxisNo.P2M2_CaCarryingUpDown1].Io.DigitalInputs.16;
arrAxisCtrl[P2AxisNo.P2M2_CaCarryingUpDown1].Io.biNegLimit:=  arrAxisCtrl[P2AxisNo.P2M2_CaCarryingUpDown1].Io.DigitalInputs.2;
arrAxisCtrl[P2AxisNo.P2M2_CaCarryingUpDown1].Io.biHomeSwitch:=arrAxisCtrl[P2AxisNo.P2M2_CaCarryingUpDown1].Io.DigitalInputs.2;

arrAxisCtrl[P2AxisNo.P2M2_CaCarryingUpDown2].Io.DigitalInputs;//二号叠台负极送片搬运2升降
arrAxisCtrl[P2AxisNo.P2M2_CaCarryingUpDown2].Io.biPosLimit:= arrAxisCtrl[P2AxisNo.P2M2_CaCarryingUpDown2].Io.DigitalInputs.16;
arrAxisCtrl[P2AxisNo.P2M2_CaCarryingUpDown2].Io.biNegLimit:=  arrAxisCtrl[P2AxisNo.P2M2_CaCarryingUpDown2].Io.DigitalInputs.2;
arrAxisCtrl[P2AxisNo.P2M2_CaCarryingUpDown2].Io.biHomeSwitch:=arrAxisCtrl[P2AxisNo.P2M2_CaCarryingUpDown2].Io.DigitalInputs.2;

arrAxisCtrl[P2AxisNo.P2M2_CaCarryingWhirling1].Io.DigitalInputs;//二号叠台负极送片搬运1旋转
arrAxisCtrl[P2AxisNo.P2M2_CaCarryingWhirling1].Io.biPosLimit:= arrAxisCtrl[P2AxisNo.P2M2_CaCarryingWhirling1].Io.DigitalInputs.16;
arrAxisCtrl[P2AxisNo.P2M2_CaCarryingWhirling1].Io.biNegLimit:=  arrAxisCtrl[P2AxisNo.P2M2_CaCarryingWhirling1].Io.DigitalInputs.2;
arrAxisCtrl[P2AxisNo.P2M2_CaCarryingWhirling1].Io.biHomeSwitch:=arrAxisCtrl[P2AxisNo.P2M2_CaCarryingWhirling1].Io.DigitalInputs.2;

arrAxisCtrl[P2AxisNo.P2M2_CadeviationX1].Io.DigitalInputs;//二号叠台负极纠偏平台X1
arrAxisCtrl[P2AxisNo.P2M2_CadeviationX1].Io.biPosLimit:= arrAxisCtrl[P2AxisNo.P2M2_CadeviationX1].Io.DigitalInputs.16;
arrAxisCtrl[P2AxisNo.P2M2_CadeviationX1].Io.biNegLimit:=  arrAxisCtrl[P2AxisNo.P2M2_CadeviationX1].Io.DigitalInputs.17;
arrAxisCtrl[P2AxisNo.P2M2_CadeviationX1].Io.biHomeSwitch:=arrAxisCtrl[P2AxisNo.P2M2_CadeviationX1].Io.DigitalInputs.2;

arrAxisCtrl[P2AxisNo.P2M2_CadeviationX2].Io.DigitalInputs;//二号叠台负极纠偏平台X2
arrAxisCtrl[P2AxisNo.P2M2_CadeviationX2].Io.biPosLimit:= arrAxisCtrl[P2AxisNo.P2M2_CadeviationX2].Io.DigitalInputs.16;
arrAxisCtrl[P2AxisNo.P2M2_CadeviationX2].Io.biNegLimit:=  arrAxisCtrl[P2AxisNo.P2M2_CadeviationX2].Io.DigitalInputs.17;
arrAxisCtrl[P2AxisNo.P2M2_CadeviationX2].Io.biHomeSwitch:=arrAxisCtrl[P2AxisNo.P2M2_CadeviationX2].Io.DigitalInputs.2;

arrAxisCtrl[P2AxisNo.P2M2_CadeviationY].Io.DigitalInputs;//二号叠台负极纠偏平台Y
arrAxisCtrl[P2AxisNo.P2M2_CadeviationY].Io.biPosLimit:= arrAxisCtrl[P2AxisNo.P2M2_CadeviationY].Io.DigitalInputs.16;
arrAxisCtrl[P2AxisNo.P2M2_CadeviationY].Io.biNegLimit:=  arrAxisCtrl[P2AxisNo.P2M2_CadeviationY].Io.DigitalInputs.17;
arrAxisCtrl[P2AxisNo.P2M2_CadeviationY].Io.biHomeSwitch:=arrAxisCtrl[P2AxisNo.P2M2_CadeviationY].Io.DigitalInputs.2;

arrAxisCtrl[P2AxisNo.P2M2_CaDTCarryingLine].Io.DigitalInputs;//二号叠台负极叠片搬运搬运//直线电机
arrAxisCtrl[P2AxisNo.P2M2_CaDTCarryingLine].Io.biPosLimit:= arrAxisCtrl[P2AxisNo.P2M2_CaDTCarryingLine].Io.DigitalInputs.17;
arrAxisCtrl[P2AxisNo.P2M2_CaDTCarryingLine].Io.biNegLimit:=  arrAxisCtrl[P2AxisNo.P2M2_CaDTCarryingLine].Io.DigitalInputs.18;
arrAxisCtrl[P2AxisNo.P2M2_CaDTCarryingLine].Io.biHomeSwitch:=arrAxisCtrl[P2AxisNo.P2M2_CaDTCarryingLine].Io.DigitalInputs.20;

arrAxisCtrl[P2AxisNo.P2M2_CaDTCarryingUpDown].Io.DigitalInputs;//二号叠台负极叠片搬运升降
arrAxisCtrl[P2AxisNo.P2M2_CaDTCarryingUpDown].Io.biPosLimit:= arrAxisCtrl[P2AxisNo.P2M2_CaDTCarryingUpDown].Io.DigitalInputs.16;
arrAxisCtrl[P2AxisNo.P2M2_CaDTCarryingUpDown].Io.biNegLimit:=  arrAxisCtrl[P2AxisNo.P2M2_CaDTCarryingUpDown].Io.DigitalInputs.2;
arrAxisCtrl[P2AxisNo.P2M2_CaDTCarryingUpDown].Io.biHomeSwitch:=arrAxisCtrl[P2AxisNo.P2M2_CaDTCarryingUpDown].Io.DigitalInputs.2;

arrAxisCtrl[P2AxisNo.P2M2_DTUpDown].Io.DigitalInputs;//二号叠台升降
arrAxisCtrl[P2AxisNo.P2M2_DTUpDown].Io.biPosLimit:= arrAxisCtrl[P2AxisNo.P2M2_DTUpDown].Io.DigitalInputs.16;
arrAxisCtrl[P2AxisNo.P2M2_DTUpDown].Io.biNegLimit:=  arrAxisCtrl[P2AxisNo.P2M2_DTUpDown].Io.DigitalInputs.2;
arrAxisCtrl[P2AxisNo.P2M2_DTUpDown].Io.biHomeSwitch:=arrAxisCtrl[P2AxisNo.P2M2_DTUpDown].Io.DigitalInputs.2;

arrAxisCtrl[P2AxisNo.P2M2_GluingLine].Io.DigitalInputs;//二号叠台侧贴胶平移
arrAxisCtrl[P2AxisNo.P2M2_GluingLine].Io.biPosLimit:= arrAxisCtrl[P2AxisNo.P2M2_GluingLine].Io.DigitalInputs.16;
arrAxisCtrl[P2AxisNo.P2M2_GluingLine].Io.biNegLimit:=  arrAxisCtrl[P2AxisNo.P2M2_GluingLine].Io.DigitalInputs.17;
arrAxisCtrl[P2AxisNo.P2M2_GluingLine].Io.biHomeSwitch:=arrAxisCtrl[P2AxisNo.P2M2_GluingLine].Io.DigitalInputs.2;

arrAxisCtrl[P2AxisNo.P2M2_GluingRetracting].Io.DigitalInputs;//二号叠台贴胶头进退
arrAxisCtrl[P2AxisNo.P2M2_GluingRetracting].Io.biPosLimit:= arrAxisCtrl[P2AxisNo.P2M2_GluingRetracting].Io.DigitalInputs.16;
arrAxisCtrl[P2AxisNo.P2M2_GluingRetracting].Io.biNegLimit:=  arrAxisCtrl[P2AxisNo.P2M2_GluingRetracting].Io.DigitalInputs.17;
arrAxisCtrl[P2AxisNo.P2M2_GluingRetracting].Io.biHomeSwitch:=arrAxisCtrl[P2AxisNo.P2M2_GluingRetracting].Io.DigitalInputs.2;

arrAxisCtrl[P2AxisNo.P2M2_GluingUpDown].Io.DigitalInputs;//二号叠台拉胶升降
arrAxisCtrl[P2AxisNo.P2M2_GluingUpDown].Io.biPosLimit:= arrAxisCtrl[P2AxisNo.P2M2_GluingUpDown].Io.DigitalInputs.16;
arrAxisCtrl[P2AxisNo.P2M2_GluingUpDown].Io.biNegLimit:=  arrAxisCtrl[P2AxisNo.P2M2_GluingUpDown].Io.DigitalInputs.17;
arrAxisCtrl[P2AxisNo.P2M2_GluingUpDown].Io.biHomeSwitch:=arrAxisCtrl[P2AxisNo.P2M2_GluingUpDown].Io.DigitalInputs.2;

arrAxisCtrl[P2AxisNo.P2M2_GluingWhirling].Io.DigitalInputs;//二号叠台贴胶夹旋转
arrAxisCtrl[P2AxisNo.P2M2_GluingWhirling].Io.biPosLimit:= arrAxisCtrl[P2AxisNo.P2M2_GluingWhirling].Io.DigitalInputs.16;
arrAxisCtrl[P2AxisNo.P2M2_GluingWhirling].Io.biNegLimit:=  arrAxisCtrl[P2AxisNo.P2M2_GluingWhirling].Io.DigitalInputs.17;
arrAxisCtrl[P2AxisNo.P2M2_GluingWhirling].Io.biHomeSwitch:=arrAxisCtrl[P2AxisNo.P2M2_GluingWhirling].Io.DigitalInputs.2;

arrAxisCtrl[P2AxisNo.P2M2_LCurlingneedleLine].Io.DigitalInputs;//二号叠台长卷针平移  雷赛
arrAxisCtrl[P2AxisNo.P2M2_LCurlingneedleLine].Io.biPosLimit:= arrAxisCtrl[P2AxisNo.P2M2_LCurlingneedleLine].Io.DigitalInputs.6;
arrAxisCtrl[P2AxisNo.P2M2_LCurlingneedleLine].Io.biNegLimit:=  arrAxisCtrl[P2AxisNo.P2M2_LCurlingneedleLine].Io.DigitalInputs.7;
arrAxisCtrl[P2AxisNo.P2M2_LCurlingneedleLine].Io.biHomeSwitch:=arrAxisCtrl[P2AxisNo.P2M2_LCurlingneedleLine].Io.DigitalInputs.7;

arrAxisCtrl[P2AxisNo.P2M2_LCurlingneedleWhirling].Io.DigitalInputs;//二号叠台长卷针旋转  雷赛
//arrAxisCtrl[P2AxisNo.P2M2_LCurlingneedleWhirling].Io.biPosLimit:=NOT arrAxisCtrl[P2AxisNo.P2M2_LCurlingneedleWhirling].Io.DigitalInputs.6;
//arrAxisCtrl[P2AxisNo.P2M2_LCurlingneedleWhirling].Io.biNegLimit:=NOT  arrAxisCtrl[P2AxisNo.P2M2_LCurlingneedleWhirling].Io.DigitalInputs.7;
arrAxisCtrl[P2AxisNo.P2M2_LCurlingneedleWhirling].Io.biHomeSwitch:=arrAxisCtrl[P2AxisNo.P2M2_LCurlingneedleWhirling].Io.DigitalInputs.2;

arrAxisCtrl[P2AxisNo.P2M2_LeftYDLine].Io.DigitalInputs;//二号叠台左压刀开合
arrAxisCtrl[P2AxisNo.P2M2_LeftYDLine].Io.biPosLimit:= arrAxisCtrl[P2AxisNo.P2M2_LeftYDLine].Io.DigitalInputs.16;
arrAxisCtrl[P2AxisNo.P2M2_LeftYDLine].Io.biNegLimit:=  arrAxisCtrl[P2AxisNo.P2M2_LeftYDLine].Io.DigitalInputs.2;
arrAxisCtrl[P2AxisNo.P2M2_LeftYDLine].Io.biHomeSwitch:=arrAxisCtrl[P2AxisNo.P2M2_LeftYDLine].Io.DigitalInputs.2;

arrAxisCtrl[P2AxisNo.P2M2_LeftYDUpDown].Io.DigitalInputs;//二号叠台左压刀升降
arrAxisCtrl[P2AxisNo.P2M2_LeftYDUpDown].Io.biPosLimit:= arrAxisCtrl[P2AxisNo.P2M2_LeftYDUpDown].Io.DigitalInputs.16;
arrAxisCtrl[P2AxisNo.P2M2_LeftYDUpDown].Io.biNegLimit:=  arrAxisCtrl[P2AxisNo.P2M2_LeftYDUpDown].Io.DigitalInputs.2;
arrAxisCtrl[P2AxisNo.P2M2_LeftYDUpDown].Io.biHomeSwitch:=arrAxisCtrl[P2AxisNo.P2M2_LeftYDUpDown].Io.DigitalInputs.2;

arrAxisCtrl[P2AxisNo.P2M2_RightYDLine].Io.DigitalInputs;//二号叠台右压刀开合
arrAxisCtrl[P2AxisNo.P2M2_RightYDLine].Io.biPosLimit:= arrAxisCtrl[P2AxisNo.P2M2_RightYDLine].Io.DigitalInputs.16;
arrAxisCtrl[P2AxisNo.P2M2_RightYDLine].Io.biNegLimit:=  arrAxisCtrl[P2AxisNo.P2M2_RightYDLine].Io.DigitalInputs.2;
arrAxisCtrl[P2AxisNo.P2M2_RightYDLine].Io.biHomeSwitch:=arrAxisCtrl[P2AxisNo.P2M2_RightYDLine].Io.DigitalInputs.2;

arrAxisCtrl[P2AxisNo.P2M2_RightYDUpDown].Io.DigitalInputs;//二号叠台右压刀升降
arrAxisCtrl[P2AxisNo.P2M2_RightYDUpDown].Io.biPosLimit:= arrAxisCtrl[P2AxisNo.P2M2_RightYDUpDown].Io.DigitalInputs.16;
arrAxisCtrl[P2AxisNo.P2M2_RightYDUpDown].Io.biNegLimit:=  arrAxisCtrl[P2AxisNo.P2M2_RightYDUpDown].Io.DigitalInputs.2;
arrAxisCtrl[P2AxisNo.P2M2_RightYDUpDown].Io.biHomeSwitch:=arrAxisCtrl[P2AxisNo.P2M2_RightYDUpDown].Io.DigitalInputs.2;

arrAxisCtrl[P2AxisNo.P2M2_SCurlingneedleLine].Io.DigitalInputs;//二号叠台短卷针平移  雷赛
arrAxisCtrl[P2AxisNo.P2M2_SCurlingneedleLine].Io.biPosLimit:= arrAxisCtrl[P2AxisNo.P2M2_SCurlingneedleLine].Io.DigitalInputs.6;
arrAxisCtrl[P2AxisNo.P2M2_SCurlingneedleLine].Io.biNegLimit:=  arrAxisCtrl[P2AxisNo.P2M2_SCurlingneedleLine].Io.DigitalInputs.7;
arrAxisCtrl[P2AxisNo.P2M2_SCurlingneedleLine].Io.biHomeSwitch:=arrAxisCtrl[P2AxisNo.P2M2_SCurlingneedleLine].Io.DigitalInputs.7;

arrAxisCtrl[P2AxisNo.P2M2_SCurlingneedleWhirling].Io.DigitalInputs;////二号叠台短卷针旋转  雷赛
//arrAxisCtrl[P2AxisNo.P2M2_SCurlingneedleWhirling].Io.biPosLimit:=NOT arrAxisCtrl[P2AxisNo.P2M2_SCurlingneedleWhirling].Io.DigitalInputs.6;
//arrAxisCtrl[P2AxisNo.P2M2_SCurlingneedleWhirling].Io.biNegLimit:=NOT  arrAxisCtrl[P2AxisNo.P2M2_SCurlingneedleWhirling].Io.DigitalInputs.7;
arrAxisCtrl[P2AxisNo.P2M2_SCurlingneedleWhirling].Io.biHomeSwitch:=arrAxisCtrl[P2AxisNo.P2M2_SCurlingneedleWhirling].Io.DigitalInputs.2;

arrAxisCtrl[P2AxisNo.P2M2_SEPTAdeviation1].Io.DigitalInputs;//二号叠台隔膜放卷纠偏
arrAxisCtrl[P2AxisNo.P2M2_SEPTAdeviation1].Io.biPosLimit:= arrAxisCtrl[P2AxisNo.P2M2_SEPTAdeviation1].Io.DigitalInputs.16;
arrAxisCtrl[P2AxisNo.P2M2_SEPTAdeviation1].Io.biNegLimit:=  arrAxisCtrl[P2AxisNo.P2M2_SEPTAdeviation1].Io.DigitalInputs.2;
arrAxisCtrl[P2AxisNo.P2M2_SEPTAdeviation1].Io.biHomeSwitch:=arrAxisCtrl[P2AxisNo.P2M2_SEPTAdeviation1].Io.DigitalInputs.2;

arrAxisCtrl[P2AxisNo.P2M2_SEPTAdeviation2].Io.DigitalInputs;//二号叠台隔膜尾部纠偏
arrAxisCtrl[P2AxisNo.P2M2_SEPTAdeviation2].Io.biPosLimit:= arrAxisCtrl[P2AxisNo.P2M2_SEPTAdeviation2].Io.DigitalInputs.16;
arrAxisCtrl[P2AxisNo.P2M2_SEPTAdeviation2].Io.biNegLimit:=  arrAxisCtrl[P2AxisNo.P2M2_SEPTAdeviation2].Io.DigitalInputs.2;
arrAxisCtrl[P2AxisNo.P2M2_SEPTAdeviation2].Io.biHomeSwitch:=arrAxisCtrl[P2AxisNo.P2M2_SEPTAdeviation2].Io.DigitalInputs.2;

arrAxisCtrl[P2AxisNo.P2M2_SEPTATCache].Io.DigitalInputs;//二号叠台隔膜缓存//直线电机
arrAxisCtrl[P2AxisNo.P2M2_SEPTATCache].Io.biPosLimit:= arrAxisCtrl[P2AxisNo.P2M2_SEPTATCache].Io.DigitalInputs.17;
arrAxisCtrl[P2AxisNo.P2M2_SEPTATCache].Io.biNegLimit:=  arrAxisCtrl[P2AxisNo.P2M2_SEPTATCache].Io.DigitalInputs.18;
arrAxisCtrl[P2AxisNo.P2M2_SEPTATCache].Io.biHomeSwitch:=arrAxisCtrl[P2AxisNo.P2M2_SEPTATCache].Io.DigitalInputs.20;

arrAxisCtrl[P2AxisNo.P2M2_SEPTATension].Io.DigitalInputs;//二号叠台隔膜摆杆张力
//arrAxisCtrl[P2AxisNo.P2M2_SEPTATension].Io.biPosLimit:=NOT arrAxisCtrl[P2AxisNo.P2M2_SEPTATension].Io.DigitalInputs.16;
//arrAxisCtrl[P2AxisNo.P2M2_SEPTATension].Io.biNegLimit:=NOT  arrAxisCtrl[P2AxisNo.P2M2_SEPTATension].Io.DigitalInputs.17;
//arrAxisCtrl[P2AxisNo.P2M2_SEPTATension].Io.biHomeSwitch:=arrAxisCtrl[P2AxisNo.P2M2_SEPTATension].Io.DigitalInputs.2;

arrAxisCtrl[P2AxisNo.P2M2_SEPTATLine].Io.DigitalInputs;//二号叠台隔膜平移//直线电机
arrAxisCtrl[P2AxisNo.P2M2_SEPTATLine].Io.biPosLimit:= arrAxisCtrl[P2AxisNo.P2M2_SEPTATLine].Io.DigitalInputs.17;
arrAxisCtrl[P2AxisNo.P2M2_SEPTATLine].Io.biNegLimit:=  arrAxisCtrl[P2AxisNo.P2M2_SEPTATLine].Io.DigitalInputs.18;
arrAxisCtrl[P2AxisNo.P2M2_SEPTATLine].Io.biHomeSwitch:=arrAxisCtrl[P2AxisNo.P2M2_SEPTATLine].Io.DigitalInputs.20;

arrAxisCtrl[P2AxisNo.P2M2_SEPTAunwinding].Io.DigitalInputs;//二号叠台隔膜放卷
//arrAxisCtrl[P2AxisNo.P2M2_SEPTAunwinding].Io.biPosLimit:=NOT arrAxisCtrl[P2AxisNo.P2M2_SEPTAunwinding].Io.DigitalInputs.16;
//arrAxisCtrl[P2AxisNo.P2M2_SEPTAunwinding].Io.biNegLimit:=NOT  arrAxisCtrl[P2AxisNo.P2M2_SEPTAunwinding].Io.DigitalInputs.17;
//arrAxisCtrl[P2AxisNo.P2M2_SEPTAunwinding].Io.biHomeSwitch:=arrAxisCtrl[P2AxisNo.P2M2_SEPTAunwinding].Io.DigitalInputs.2;

arrAxisCtrl[P2AxisNo.P2M2_TailCurlLine].Io.DigitalInputs;//二号叠台尾卷夹电芯平移
arrAxisCtrl[P2AxisNo.P2M2_TailCurlLine].Io.biPosLimit:= arrAxisCtrl[P2AxisNo.P2M2_TailCurlLine].Io.DigitalInputs.16;
arrAxisCtrl[P2AxisNo.P2M2_TailCurlLine].Io.biNegLimit:=  arrAxisCtrl[P2AxisNo.P2M2_TailCurlLine].Io.DigitalInputs.17;
arrAxisCtrl[P2AxisNo.P2M2_TailCurlLine].Io.biHomeSwitch:=arrAxisCtrl[P2AxisNo.P2M2_TailCurlLine].Io.DigitalInputs.2;

arrAxisCtrl[P2AxisNo.P2M2_TailCurlRetracting].Io.DigitalInputs;//二号叠台尾卷夹电芯伸缩
arrAxisCtrl[P2AxisNo.P2M2_TailCurlRetracting].Io.biPosLimit:= arrAxisCtrl[P2AxisNo.P2M2_TailCurlRetracting].Io.DigitalInputs.16;
arrAxisCtrl[P2AxisNo.P2M2_TailCurlRetracting].Io.biNegLimit:=  arrAxisCtrl[P2AxisNo.P2M2_TailCurlRetracting].Io.DigitalInputs.17;
arrAxisCtrl[P2AxisNo.P2M2_TailCurlRetracting].Io.biHomeSwitch:=arrAxisCtrl[P2AxisNo.P2M2_TailCurlRetracting].Io.DigitalInputs.17;

arrAxisCtrl[P2AxisNo.P2M2_TailCurlSEPTALine].Io.DigitalInputs;//二号叠台夹膜平移
arrAxisCtrl[P2AxisNo.P2M2_TailCurlSEPTALine].Io.biPosLimit:= arrAxisCtrl[P2AxisNo.P2M2_TailCurlSEPTALine].Io.DigitalInputs.16;
arrAxisCtrl[P2AxisNo.P2M2_TailCurlSEPTALine].Io.biNegLimit:=  arrAxisCtrl[P2AxisNo.P2M2_TailCurlSEPTALine].Io.DigitalInputs.17;
arrAxisCtrl[P2AxisNo.P2M2_TailCurlSEPTALine].Io.biHomeSwitch:=arrAxisCtrl[P2AxisNo.P2M2_TailCurlSEPTALine].Io.DigitalInputs.17;

arrAxisCtrl[P2AxisNo.P2M2_TailCurlSEPTAUpDown].Io.DigitalInputs;//二号叠台夹膜升降
arrAxisCtrl[P2AxisNo.P2M2_TailCurlSEPTAUpDown].Io.biPosLimit:= arrAxisCtrl[P2AxisNo.P2M2_TailCurlSEPTAUpDown].Io.DigitalInputs.16;
arrAxisCtrl[P2AxisNo.P2M2_TailCurlSEPTAUpDown].Io.biNegLimit:=  arrAxisCtrl[P2AxisNo.P2M2_TailCurlSEPTAUpDown].Io.DigitalInputs.2;
arrAxisCtrl[P2AxisNo.P2M2_TailCurlSEPTAUpDown].Io.biHomeSwitch:=arrAxisCtrl[P2AxisNo.P2M2_TailCurlSEPTAUpDown].Io.DigitalInputs.2;

arrAxisCtrl[P2AxisNo.P2M2_TailCurlUpDown].Io.DigitalInputs;//二号叠台尾卷夹电芯升降
arrAxisCtrl[P2AxisNo.P2M2_TailCurlUpDown].Io.biPosLimit:= arrAxisCtrl[P2AxisNo.P2M2_TailCurlUpDown].Io.DigitalInputs.16;
arrAxisCtrl[P2AxisNo.P2M2_TailCurlUpDown].Io.biNegLimit:=  arrAxisCtrl[P2AxisNo.P2M2_TailCurlUpDown].Io.DigitalInputs.17;
arrAxisCtrl[P2AxisNo.P2M2_TailCurlUpDown].Io.biHomeSwitch:=arrAxisCtrl[P2AxisNo.P2M2_TailCurlUpDown].Io.DigitalInputs.2;

arrAxisCtrl[P2AxisNo.P2M2_TailCurlWhirling].Io.DigitalInputs;//二号叠台尾卷夹电芯旋转
arrAxisCtrl[P2AxisNo.P2M2_TailCurlWhirling].Io.biPosLimit:= arrAxisCtrl[P2AxisNo.P2M2_TailCurlWhirling].Io.DigitalInputs.16;
arrAxisCtrl[P2AxisNo.P2M2_TailCurlWhirling].Io.biNegLimit:=  arrAxisCtrl[P2AxisNo.P2M2_TailCurlWhirling].Io.DigitalInputs.17;
arrAxisCtrl[P2AxisNo.P2M2_TailCurlWhirling].Io.biHomeSwitch:=arrAxisCtrl[P2AxisNo.P2M2_TailCurlWhirling].Io.DigitalInputs.17;








//3叠台
arrAxisCtrl[P2AxisNo.P2M3_AnCarryingLine].Io.DigitalInputs;//三号叠台正极送片搬运平移//直线电机
arrAxisCtrl[P2AxisNo.P2M3_AnCarryingLine].Io.biPosLimit:= arrAxisCtrl[P2AxisNo.P2M3_AnCarryingLine].Io.DigitalInputs.17;
arrAxisCtrl[P2AxisNo.P2M3_AnCarryingLine].Io.biNegLimit:=  arrAxisCtrl[P2AxisNo.P2M3_AnCarryingLine].Io.DigitalInputs.18;
arrAxisCtrl[P2AxisNo.P2M3_AnCarryingLine].Io.biHomeSwitch:=arrAxisCtrl[P2AxisNo.P2M3_AnCarryingLine].Io.DigitalInputs.20;

arrAxisCtrl[P2AxisNo.P2M3_AnCarryingUpDown].Io.DigitalInputs;//三号叠台正极送片搬运升降
arrAxisCtrl[P2AxisNo.P2M3_AnCarryingUpDown].Io.biPosLimit:= arrAxisCtrl[P2AxisNo.P2M3_AnCarryingUpDown].Io.DigitalInputs.16;
arrAxisCtrl[P2AxisNo.P2M3_AnCarryingUpDown].Io.biNegLimit:=  arrAxisCtrl[P2AxisNo.P2M3_AnCarryingUpDown].Io.DigitalInputs.2;
arrAxisCtrl[P2AxisNo.P2M3_AnCarryingUpDown].Io.biHomeSwitch:=arrAxisCtrl[P2AxisNo.P2M3_AnCarryingUpDown].Io.DigitalInputs.2;

arrAxisCtrl[P2AxisNo.P2M3_AnCarryingWhirling].Io.DigitalInputs;//三号叠台正极送片搬运旋转
arrAxisCtrl[P2AxisNo.P2M3_AnCarryingWhirling].Io.biPosLimit:= arrAxisCtrl[P2AxisNo.P2M3_AnCarryingWhirling].Io.DigitalInputs.16;
arrAxisCtrl[P2AxisNo.P2M3_AnCarryingWhirling].Io.biNegLimit:=  arrAxisCtrl[P2AxisNo.P2M3_AnCarryingWhirling].Io.DigitalInputs.2;
arrAxisCtrl[P2AxisNo.P2M3_AnCarryingWhirling].Io.biHomeSwitch:=arrAxisCtrl[P2AxisNo.P2M3_AnCarryingWhirling].Io.DigitalInputs.2;

arrAxisCtrl[P2AxisNo.P2M3_AndeviationX1].Io.DigitalInputs;//三号叠台正极纠偏平台X1
arrAxisCtrl[P2AxisNo.P2M3_AndeviationX1].Io.biPosLimit:= arrAxisCtrl[P2AxisNo.P2M3_AndeviationX1].Io.DigitalInputs.16;
arrAxisCtrl[P2AxisNo.P2M3_AndeviationX1].Io.biNegLimit:=  arrAxisCtrl[P2AxisNo.P2M3_AndeviationX1].Io.DigitalInputs.17;
arrAxisCtrl[P2AxisNo.P2M3_AndeviationX1].Io.biHomeSwitch:=arrAxisCtrl[P2AxisNo.P2M3_AndeviationX1].Io.DigitalInputs.2;

arrAxisCtrl[P2AxisNo.P2M3_AndeviationX2].Io.DigitalInputs;//三号叠台正极纠偏平台X2
arrAxisCtrl[P2AxisNo.P2M3_AndeviationX2].Io.biPosLimit:= arrAxisCtrl[P2AxisNo.P2M3_AndeviationX2].Io.DigitalInputs.16;
arrAxisCtrl[P2AxisNo.P2M3_AndeviationX2].Io.biNegLimit:=  arrAxisCtrl[P2AxisNo.P2M3_AndeviationX2].Io.DigitalInputs.17;
arrAxisCtrl[P2AxisNo.P2M3_AndeviationX2].Io.biHomeSwitch:=arrAxisCtrl[P2AxisNo.P2M3_AndeviationX2].Io.DigitalInputs.2;

arrAxisCtrl[P2AxisNo.P2M3_AndeviationY].Io.DigitalInputs;//三号叠台正极纠偏平台Y
arrAxisCtrl[P2AxisNo.P2M3_AndeviationY].Io.biPosLimit:= arrAxisCtrl[P2AxisNo.P2M3_AndeviationY].Io.DigitalInputs.16;
arrAxisCtrl[P2AxisNo.P2M3_AndeviationY].Io.biNegLimit:=  arrAxisCtrl[P2AxisNo.P2M3_AndeviationY].Io.DigitalInputs.17;
arrAxisCtrl[P2AxisNo.P2M3_AndeviationY].Io.biHomeSwitch:=arrAxisCtrl[P2AxisNo.P2M3_AndeviationY].Io.DigitalInputs.2;

arrAxisCtrl[P2AxisNo.P2M3_AnDTCarryingLine].Io.DigitalInputs;//三号叠台正极叠台搬运平移//直线电机
arrAxisCtrl[P2AxisNo.P2M3_AnDTCarryingLine].Io.biPosLimit:= arrAxisCtrl[P2AxisNo.P2M3_AnDTCarryingLine].Io.DigitalInputs.17;
arrAxisCtrl[P2AxisNo.P2M3_AnDTCarryingLine].Io.biNegLimit:=  arrAxisCtrl[P2AxisNo.P2M3_AnDTCarryingLine].Io.DigitalInputs.18;
arrAxisCtrl[P2AxisNo.P2M3_AnDTCarryingLine].Io.biHomeSwitch:=arrAxisCtrl[P2AxisNo.P2M3_AnDTCarryingLine].Io.DigitalInputs.20;

arrAxisCtrl[P2AxisNo.P2M3_AnDTCarryingUpDown].Io.DigitalInputs;//三号叠台正极叠台搬运升降
arrAxisCtrl[P2AxisNo.P2M3_AnDTCarryingUpDown].Io.biPosLimit:= arrAxisCtrl[P2AxisNo.P2M3_AnDTCarryingUpDown].Io.DigitalInputs.16;
arrAxisCtrl[P2AxisNo.P2M3_AnDTCarryingUpDown].Io.biNegLimit:=  arrAxisCtrl[P2AxisNo.P2M3_AnDTCarryingUpDown].Io.DigitalInputs.2;
arrAxisCtrl[P2AxisNo.P2M3_AnDTCarryingUpDown].Io.biHomeSwitch:=arrAxisCtrl[P2AxisNo.P2M3_AnDTCarryingUpDown].Io.DigitalInputs.2;

arrAxisCtrl[P2AxisNo.P2M3_CaBelt].Io.DigitalInputs;//三号叠台负极送片皮带
//arrAxisCtrl[P2AxisNo.P2M3_CaBelt].Io.biPosLimit:=NOT arrAxisCtrl[P2AxisNo.P2M3_CaBelt].Io.DigitalInputs.16;
//arrAxisCtrl[P2AxisNo.P2M3_CaBelt].Io.biNegLimit:=NOT  arrAxisCtrl[P2AxisNo.P2M3_CaBelt].Io.DigitalInputs.17;
//arrAxisCtrl[P2AxisNo.P2M3_CaBelt].Io.biHomeSwitch:=arrAxisCtrl[P2AxisNo.P2M3_CaBelt].Io.DigitalInputs.2;

arrAxisCtrl[P2AxisNo.P2M3_CaCarryingLine1].Io.DigitalInputs;//三号叠台负极搬运1平移//直线电机
arrAxisCtrl[P2AxisNo.P2M3_CaCarryingLine1].Io.biPosLimit:= arrAxisCtrl[P2AxisNo.P2M3_CaCarryingLine1].Io.DigitalInputs.17;
arrAxisCtrl[P2AxisNo.P2M3_CaCarryingLine1].Io.biNegLimit:=  arrAxisCtrl[P2AxisNo.P2M3_CaCarryingLine1].Io.DigitalInputs.18;
arrAxisCtrl[P2AxisNo.P2M3_CaCarryingLine1].Io.biHomeSwitch:=arrAxisCtrl[P2AxisNo.P2M3_CaCarryingLine1].Io.DigitalInputs.20;

arrAxisCtrl[P2AxisNo.P2M3_CaCarryingLine2].Io.DigitalInputs;//三号叠台负极搬运2平移//直线电机
arrAxisCtrl[P2AxisNo.P2M3_CaCarryingLine2].Io.biPosLimit:= arrAxisCtrl[P2AxisNo.P2M3_CaCarryingLine2].Io.DigitalInputs.17;
arrAxisCtrl[P2AxisNo.P2M3_CaCarryingLine2].Io.biNegLimit:=  arrAxisCtrl[P2AxisNo.P2M3_CaCarryingLine2].Io.DigitalInputs.18;
arrAxisCtrl[P2AxisNo.P2M3_CaCarryingLine2].Io.biHomeSwitch:=arrAxisCtrl[P2AxisNo.P2M3_CaCarryingLine2].Io.DigitalInputs.20;

arrAxisCtrl[P2AxisNo.P2M3_CaCarryingUpDown1].Io.DigitalInputs;//三号叠台负极搬运1升降
arrAxisCtrl[P2AxisNo.P2M3_CaCarryingUpDown1].Io.biPosLimit:= arrAxisCtrl[P2AxisNo.P2M3_CaCarryingUpDown1].Io.DigitalInputs.16;
arrAxisCtrl[P2AxisNo.P2M3_CaCarryingUpDown1].Io.biNegLimit:=  arrAxisCtrl[P2AxisNo.P2M3_CaCarryingUpDown1].Io.DigitalInputs.2;
arrAxisCtrl[P2AxisNo.P2M3_CaCarryingUpDown1].Io.biHomeSwitch:=arrAxisCtrl[P2AxisNo.P2M3_CaCarryingUpDown1].Io.DigitalInputs.2;

arrAxisCtrl[P2AxisNo.P2M3_CaCarryingUpDown2].Io.DigitalInputs;//三号叠台负送片搬运2升降
arrAxisCtrl[P2AxisNo.P2M3_CaCarryingUpDown2].Io.biPosLimit:= arrAxisCtrl[P2AxisNo.P2M3_CaCarryingUpDown2].Io.DigitalInputs.16;
arrAxisCtrl[P2AxisNo.P2M3_CaCarryingUpDown2].Io.biNegLimit:=  arrAxisCtrl[P2AxisNo.P2M3_CaCarryingUpDown2].Io.DigitalInputs.2;
arrAxisCtrl[P2AxisNo.P2M3_CaCarryingUpDown2].Io.biHomeSwitch:=arrAxisCtrl[P2AxisNo.P2M3_CaCarryingUpDown2].Io.DigitalInputs.2;

arrAxisCtrl[P2AxisNo.P2M3_CaCarryingWhirling1].Io.DigitalInputs;//三号叠台负极搬运1旋转
arrAxisCtrl[P2AxisNo.P2M3_CaCarryingWhirling1].Io.biPosLimit:= arrAxisCtrl[P2AxisNo.P2M3_CaCarryingWhirling1].Io.DigitalInputs.16;
arrAxisCtrl[P2AxisNo.P2M3_CaCarryingWhirling1].Io.biNegLimit:=  arrAxisCtrl[P2AxisNo.P2M3_CaCarryingWhirling1].Io.DigitalInputs.2;
arrAxisCtrl[P2AxisNo.P2M3_CaCarryingWhirling1].Io.biHomeSwitch:=arrAxisCtrl[P2AxisNo.P2M3_CaCarryingWhirling1].Io.DigitalInputs.2;

arrAxisCtrl[P2AxisNo.P2M3_CadeviationX1].Io.DigitalInputs;//三号叠台负极纠偏平台X1
arrAxisCtrl[P2AxisNo.P2M3_CadeviationX1].Io.biPosLimit:= arrAxisCtrl[P2AxisNo.P2M3_CadeviationX1].Io.DigitalInputs.16;
arrAxisCtrl[P2AxisNo.P2M3_CadeviationX1].Io.biNegLimit:=  arrAxisCtrl[P2AxisNo.P2M3_CadeviationX1].Io.DigitalInputs.17;
arrAxisCtrl[P2AxisNo.P2M3_CadeviationX1].Io.biHomeSwitch:=arrAxisCtrl[P2AxisNo.P2M3_CadeviationX1].Io.DigitalInputs.2;

arrAxisCtrl[P2AxisNo.P2M3_CadeviationX2].Io.DigitalInputs;//三号叠台负极纠偏平台X2
arrAxisCtrl[P2AxisNo.P2M3_CadeviationX2].Io.biPosLimit:= arrAxisCtrl[P2AxisNo.P2M3_CadeviationX2].Io.DigitalInputs.16;
arrAxisCtrl[P2AxisNo.P2M3_CadeviationX2].Io.biNegLimit:=  arrAxisCtrl[P2AxisNo.P2M3_CadeviationX2].Io.DigitalInputs.17;
arrAxisCtrl[P2AxisNo.P2M3_CadeviationX2].Io.biHomeSwitch:=arrAxisCtrl[P2AxisNo.P2M3_CadeviationX2].Io.DigitalInputs.2;

arrAxisCtrl[P2AxisNo.P2M3_CadeviationY].Io.DigitalInputs;//三号叠台负极纠偏平台Y
arrAxisCtrl[P2AxisNo.P2M3_CadeviationY].Io.biPosLimit:= arrAxisCtrl[P2AxisNo.P2M3_CadeviationY].Io.DigitalInputs.16;
arrAxisCtrl[P2AxisNo.P2M3_CadeviationY].Io.biNegLimit:=  arrAxisCtrl[P2AxisNo.P2M3_CadeviationY].Io.DigitalInputs.17;
arrAxisCtrl[P2AxisNo.P2M3_CadeviationY].Io.biHomeSwitch:=arrAxisCtrl[P2AxisNo.P2M3_CadeviationY].Io.DigitalInputs.2;

arrAxisCtrl[P2AxisNo.P2M3_CaDTCarryingLine].Io.DigitalInputs;//三号叠台负极叠片搬运平移//直线电机
arrAxisCtrl[P2AxisNo.P2M3_CaDTCarryingLine].Io.biPosLimit:= arrAxisCtrl[P2AxisNo.P2M3_CaDTCarryingLine].Io.DigitalInputs.17;
arrAxisCtrl[P2AxisNo.P2M3_CaDTCarryingLine].Io.biNegLimit:=  arrAxisCtrl[P2AxisNo.P2M3_CaDTCarryingLine].Io.DigitalInputs.18;
arrAxisCtrl[P2AxisNo.P2M3_CaDTCarryingLine].Io.biHomeSwitch:=arrAxisCtrl[P2AxisNo.P2M3_CaDTCarryingLine].Io.DigitalInputs.20;

arrAxisCtrl[P2AxisNo.P2M3_CaDTCarryingUpDown].Io.DigitalInputs;//负极叠台搬运升降
arrAxisCtrl[P2AxisNo.P2M3_CaDTCarryingUpDown].Io.biPosLimit:= arrAxisCtrl[P2AxisNo.P2M3_CaDTCarryingUpDown].Io.DigitalInputs.16;
arrAxisCtrl[P2AxisNo.P2M3_CaDTCarryingUpDown].Io.biNegLimit:=  arrAxisCtrl[P2AxisNo.P2M3_CaDTCarryingUpDown].Io.DigitalInputs.2;
arrAxisCtrl[P2AxisNo.P2M3_CaDTCarryingUpDown].Io.biHomeSwitch:=arrAxisCtrl[P2AxisNo.P2M3_CaDTCarryingUpDown].Io.DigitalInputs.2;

arrAxisCtrl[P2AxisNo.P2M3_DTUpDown].Io.DigitalInputs;//三号叠台叠台升降
arrAxisCtrl[P2AxisNo.P2M3_DTUpDown].Io.biPosLimit:= arrAxisCtrl[P2AxisNo.P2M3_DTUpDown].Io.DigitalInputs.16;
arrAxisCtrl[P2AxisNo.P2M3_DTUpDown].Io.biNegLimit:=  arrAxisCtrl[P2AxisNo.P2M3_DTUpDown].Io.DigitalInputs.2;
arrAxisCtrl[P2AxisNo.P2M3_DTUpDown].Io.biHomeSwitch:=arrAxisCtrl[P2AxisNo.P2M3_DTUpDown].Io.DigitalInputs.2;

arrAxisCtrl[P2AxisNo.P2M3_GluingLine].Io.DigitalInputs;//三号叠台侧贴胶夹平移
arrAxisCtrl[P2AxisNo.P2M3_GluingLine].Io.biPosLimit:= arrAxisCtrl[P2AxisNo.P2M3_GluingLine].Io.DigitalInputs.16;
arrAxisCtrl[P2AxisNo.P2M3_GluingLine].Io.biNegLimit:=  arrAxisCtrl[P2AxisNo.P2M3_GluingLine].Io.DigitalInputs.17;
arrAxisCtrl[P2AxisNo.P2M3_GluingLine].Io.biHomeSwitch:=arrAxisCtrl[P2AxisNo.P2M3_GluingLine].Io.DigitalInputs.2;

arrAxisCtrl[P2AxisNo.P2M3_GluingRetracting].Io.DigitalInputs;//三号叠台侧贴胶夹进退
arrAxisCtrl[P2AxisNo.P2M3_GluingRetracting].Io.biPosLimit:= arrAxisCtrl[P2AxisNo.P2M3_GluingRetracting].Io.DigitalInputs.16;
arrAxisCtrl[P2AxisNo.P2M3_GluingRetracting].Io.biNegLimit:=  arrAxisCtrl[P2AxisNo.P2M3_GluingRetracting].Io.DigitalInputs.17;
arrAxisCtrl[P2AxisNo.P2M3_GluingRetracting].Io.biHomeSwitch:=arrAxisCtrl[P2AxisNo.P2M3_GluingRetracting].Io.DigitalInputs.2;

arrAxisCtrl[P2AxisNo.P2M3_GluingUpDown].Io.DigitalInputs;//三号叠台拉胶升降
arrAxisCtrl[P2AxisNo.P2M3_GluingUpDown].Io.biPosLimit:= arrAxisCtrl[P2AxisNo.P2M3_GluingUpDown].Io.DigitalInputs.16;
arrAxisCtrl[P2AxisNo.P2M3_GluingUpDown].Io.biNegLimit:=  arrAxisCtrl[P2AxisNo.P2M3_GluingUpDown].Io.DigitalInputs.17;
arrAxisCtrl[P2AxisNo.P2M3_GluingUpDown].Io.biHomeSwitch:=arrAxisCtrl[P2AxisNo.P2M3_GluingUpDown].Io.DigitalInputs.2;

arrAxisCtrl[P2AxisNo.P2M3_GluingWhirling].Io.DigitalInputs;//三号叠台侧胶夹旋转
arrAxisCtrl[P2AxisNo.P2M3_GluingWhirling].Io.biPosLimit:= arrAxisCtrl[P2AxisNo.P2M3_GluingWhirling].Io.DigitalInputs.16;
arrAxisCtrl[P2AxisNo.P2M3_GluingWhirling].Io.biNegLimit:=  arrAxisCtrl[P2AxisNo.P2M3_GluingWhirling].Io.DigitalInputs.17;
arrAxisCtrl[P2AxisNo.P2M3_GluingWhirling].Io.biHomeSwitch:=arrAxisCtrl[P2AxisNo.P2M3_GluingWhirling].Io.DigitalInputs.2;

arrAxisCtrl[P2AxisNo.P2M3_LCurlingneedleLine].Io.DigitalInputs;//三号叠台长卷针平移   雷赛
arrAxisCtrl[P2AxisNo.P2M3_LCurlingneedleLine].Io.biPosLimit:= arrAxisCtrl[P2AxisNo.P2M3_LCurlingneedleLine].Io.DigitalInputs.6;
arrAxisCtrl[P2AxisNo.P2M3_LCurlingneedleLine].Io.biNegLimit:=  arrAxisCtrl[P2AxisNo.P2M3_LCurlingneedleLine].Io.DigitalInputs.7;
arrAxisCtrl[P2AxisNo.P2M3_LCurlingneedleLine].Io.biHomeSwitch:=arrAxisCtrl[P2AxisNo.P2M3_LCurlingneedleLine].Io.DigitalInputs.7;

arrAxisCtrl[P2AxisNo.P2M3_LCurlingneedleWhirling].Io.DigitalInputs;//三号叠台长卷针旋转  雷赛
//arrAxisCtrl[P2AxisNo.P2M3_LCurlingneedleWhirling].Io.biPosLimit:=NOT arrAxisCtrl[P2AxisNo.P2M3_LCurlingneedleWhirling].Io.DigitalInputs.6;
//arrAxisCtrl[P2AxisNo.P2M3_LCurlingneedleWhirling].Io.biNegLimit:=NOT  arrAxisCtrl[P2AxisNo.P2M3_LCurlingneedleWhirling].Io.DigitalInputs.7;
arrAxisCtrl[P2AxisNo.P2M3_LCurlingneedleWhirling].Io.biHomeSwitch:=arrAxisCtrl[P2AxisNo.P2M3_LCurlingneedleWhirling].Io.DigitalInputs.2;

arrAxisCtrl[P2AxisNo.P2M3_LeftYDLine].Io.DigitalInputs;//三号叠台左压刀开合
arrAxisCtrl[P2AxisNo.P2M3_LeftYDLine].Io.biPosLimit:= arrAxisCtrl[P2AxisNo.P2M3_LeftYDLine].Io.DigitalInputs.16;
arrAxisCtrl[P2AxisNo.P2M3_LeftYDLine].Io.biNegLimit:=  arrAxisCtrl[P2AxisNo.P2M3_LeftYDLine].Io.DigitalInputs.2;
arrAxisCtrl[P2AxisNo.P2M3_LeftYDLine].Io.biHomeSwitch:=arrAxisCtrl[P2AxisNo.P2M3_LeftYDLine].Io.DigitalInputs.2;

arrAxisCtrl[P2AxisNo.P2M3_LeftYDUpDown].Io.DigitalInputs;//三号叠台左压刀升降
arrAxisCtrl[P2AxisNo.P2M3_LeftYDUpDown].Io.biPosLimit:= arrAxisCtrl[P2AxisNo.P2M3_LeftYDUpDown].Io.DigitalInputs.16;
arrAxisCtrl[P2AxisNo.P2M3_LeftYDUpDown].Io.biNegLimit:=  arrAxisCtrl[P2AxisNo.P2M3_LeftYDUpDown].Io.DigitalInputs.2;
arrAxisCtrl[P2AxisNo.P2M3_LeftYDUpDown].Io.biHomeSwitch:=arrAxisCtrl[P2AxisNo.P2M3_LeftYDUpDown].Io.DigitalInputs.2;

arrAxisCtrl[P2AxisNo.P2M3_RightYDLine].Io.DigitalInputs;//三号叠台右压刀开合
arrAxisCtrl[P2AxisNo.P2M3_RightYDLine].Io.biPosLimit:= arrAxisCtrl[P2AxisNo.P2M3_RightYDLine].Io.DigitalInputs.16;
arrAxisCtrl[P2AxisNo.P2M3_RightYDLine].Io.biNegLimit:=  arrAxisCtrl[P2AxisNo.P2M3_RightYDLine].Io.DigitalInputs.2;
arrAxisCtrl[P2AxisNo.P2M3_RightYDLine].Io.biHomeSwitch:=arrAxisCtrl[P2AxisNo.P2M3_RightYDLine].Io.DigitalInputs.2;

arrAxisCtrl[P2AxisNo.P2M3_RightYDUpDown].Io.DigitalInputs;//三号叠台右压刀升降
arrAxisCtrl[P2AxisNo.P2M3_RightYDUpDown].Io.biPosLimit:= arrAxisCtrl[P2AxisNo.P2M3_RightYDUpDown].Io.DigitalInputs.16;
arrAxisCtrl[P2AxisNo.P2M3_RightYDUpDown].Io.biNegLimit:=  arrAxisCtrl[P2AxisNo.P2M3_RightYDUpDown].Io.DigitalInputs.2;
arrAxisCtrl[P2AxisNo.P2M3_RightYDUpDown].Io.biHomeSwitch:=arrAxisCtrl[P2AxisNo.P2M3_RightYDUpDown].Io.DigitalInputs.2;

arrAxisCtrl[P2AxisNo.P2M3_SCurlingneedleLine].Io.DigitalInputs;//三号叠台短卷针平移   雷赛
arrAxisCtrl[P2AxisNo.P2M3_SCurlingneedleLine].Io.biPosLimit:= arrAxisCtrl[P2AxisNo.P2M3_SCurlingneedleLine].Io.DigitalInputs.6;
arrAxisCtrl[P2AxisNo.P2M3_SCurlingneedleLine].Io.biNegLimit:=  arrAxisCtrl[P2AxisNo.P2M3_SCurlingneedleLine].Io.DigitalInputs.7;
arrAxisCtrl[P2AxisNo.P2M3_SCurlingneedleLine].Io.biHomeSwitch:=arrAxisCtrl[P2AxisNo.P2M3_SCurlingneedleLine].Io.DigitalInputs.7;

arrAxisCtrl[P2AxisNo.P2M3_SCurlingneedleWhirling].Io.DigitalInputs;//三号叠台短卷针旋转
//arrAxisCtrl[P2AxisNo.P2M3_SCurlingneedleWhirling].Io.biPosLimit:=NOT arrAxisCtrl[P2AxisNo.P2M3_SCurlingneedleWhirling].Io.DigitalInputs.6;
//arrAxisCtrl[P2AxisNo.P2M3_SCurlingneedleWhirling].Io.biNegLimit:=NOT  arrAxisCtrl[P2AxisNo.P2M3_SCurlingneedleWhirling].Io.DigitalInputs.7;
arrAxisCtrl[P2AxisNo.P2M3_SCurlingneedleWhirling].Io.biHomeSwitch:=arrAxisCtrl[P2AxisNo.P2M3_SCurlingneedleWhirling].Io.DigitalInputs.2;

arrAxisCtrl[P2AxisNo.P2M3_SEPTAdeviation1].Io.DigitalInputs;//三号叠台隔膜放卷纠偏
arrAxisCtrl[P2AxisNo.P2M3_SEPTAdeviation1].Io.biPosLimit:= arrAxisCtrl[P2AxisNo.P2M3_SEPTAdeviation1].Io.DigitalInputs.16;
arrAxisCtrl[P2AxisNo.P2M3_SEPTAdeviation1].Io.biNegLimit:=  arrAxisCtrl[P2AxisNo.P2M3_SEPTAdeviation1].Io.DigitalInputs.2;
arrAxisCtrl[P2AxisNo.P2M3_SEPTAdeviation1].Io.biHomeSwitch:=arrAxisCtrl[P2AxisNo.P2M3_SEPTAdeviation1].Io.DigitalInputs.2;

arrAxisCtrl[P2AxisNo.P2M3_SEPTAdeviation2].Io.DigitalInputs;//三号叠台隔膜尾部纠偏
arrAxisCtrl[P2AxisNo.P2M3_SEPTAdeviation2].Io.biPosLimit:= arrAxisCtrl[P2AxisNo.P2M3_SEPTAdeviation2].Io.DigitalInputs.16;
arrAxisCtrl[P2AxisNo.P2M3_SEPTAdeviation2].Io.biNegLimit:=  arrAxisCtrl[P2AxisNo.P2M3_SEPTAdeviation2].Io.DigitalInputs.2;
arrAxisCtrl[P2AxisNo.P2M3_SEPTAdeviation2].Io.biHomeSwitch:=arrAxisCtrl[P2AxisNo.P2M3_SEPTAdeviation2].Io.DigitalInputs.2;

arrAxisCtrl[P2AxisNo.P2M3_SEPTATCache].Io.DigitalInputs;//三号叠台隔膜缓存//直线电机
arrAxisCtrl[P2AxisNo.P2M3_SEPTATCache].Io.biPosLimit:= arrAxisCtrl[P2AxisNo.P2M3_SEPTATCache].Io.DigitalInputs.17;
arrAxisCtrl[P2AxisNo.P2M3_SEPTATCache].Io.biNegLimit:=  arrAxisCtrl[P2AxisNo.P2M3_SEPTATCache].Io.DigitalInputs.18;
arrAxisCtrl[P2AxisNo.P2M3_SEPTATCache].Io.biHomeSwitch:=arrAxisCtrl[P2AxisNo.P2M3_SEPTATCache].Io.DigitalInputs.20;

arrAxisCtrl[P2AxisNo.P2M3_SEPTATension].Io.DigitalInputs;////三号叠台隔膜摆杆张力
//arrAxisCtrl[P2AxisNo.P2M3_SEPTATension].Io.biPosLimit:=NOT arrAxisCtrl[P2AxisNo.P2M3_SEPTATension].Io.DigitalInputs.16;
//arrAxisCtrl[P2AxisNo.P2M3_SEPTATension].Io.biNegLimit:=NOT  arrAxisCtrl[P2AxisNo.P2M3_SEPTATension].Io.DigitalInputs.17;
//arrAxisCtrl[P2AxisNo.P2M3_SEPTATension].Io.biHomeSwitch:=arrAxisCtrl[P2AxisNo.P2M3_SEPTATension].Io.DigitalInputs.2;

arrAxisCtrl[P2AxisNo.P2M3_SEPTATLine].Io.DigitalInputs;//三号叠台隔膜平移//直线电机
arrAxisCtrl[P2AxisNo.P2M3_SEPTATLine].Io.biPosLimit:= arrAxisCtrl[P2AxisNo.P2M3_SEPTATLine].Io.DigitalInputs.17;
arrAxisCtrl[P2AxisNo.P2M3_SEPTATLine].Io.biNegLimit:=  arrAxisCtrl[P2AxisNo.P2M3_SEPTATLine].Io.DigitalInputs.18;
arrAxisCtrl[P2AxisNo.P2M3_SEPTATLine].Io.biHomeSwitch:=arrAxisCtrl[P2AxisNo.P2M3_SEPTATLine].Io.DigitalInputs.20;

arrAxisCtrl[P2AxisNo.P2M3_SEPTAunwinding].Io.DigitalInputs;//三号叠台隔膜放卷
//arrAxisCtrl[P2AxisNo.P2M3_SEPTAunwinding].Io.biPosLimit:=NOT arrAxisCtrl[P2AxisNo.P2M3_SEPTAunwinding].Io.DigitalInputs.16;
//arrAxisCtrl[P2AxisNo.P2M3_SEPTAunwinding].Io.biNegLimit:=NOT  arrAxisCtrl[P2AxisNo.P2M3_SEPTAunwinding].Io.DigitalInputs.17;
//arrAxisCtrl[P2AxisNo.P2M3_SEPTAunwinding].Io.biHomeSwitch:=arrAxisCtrl[P2AxisNo.P2M3_SEPTAunwinding].Io.DigitalInputs.2;

arrAxisCtrl[P2AxisNo.P2M3_TailCurlLine].Io.DigitalInputs;//三号叠台尾卷电芯平移
arrAxisCtrl[P2AxisNo.P2M3_TailCurlLine].Io.biPosLimit:= arrAxisCtrl[P2AxisNo.P2M3_TailCurlLine].Io.DigitalInputs.16;
arrAxisCtrl[P2AxisNo.P2M3_TailCurlLine].Io.biNegLimit:=  arrAxisCtrl[P2AxisNo.P2M3_TailCurlLine].Io.DigitalInputs.17;
arrAxisCtrl[P2AxisNo.P2M3_TailCurlLine].Io.biHomeSwitch:=arrAxisCtrl[P2AxisNo.P2M3_TailCurlLine].Io.DigitalInputs.2;

arrAxisCtrl[P2AxisNo.P2M3_TailCurlRetracting].Io.DigitalInputs;//三号叠台尾卷夹电芯伸缩
arrAxisCtrl[P2AxisNo.P2M3_TailCurlRetracting].Io.biPosLimit:= arrAxisCtrl[P2AxisNo.P2M3_TailCurlRetracting].Io.DigitalInputs.16;
arrAxisCtrl[P2AxisNo.P2M3_TailCurlRetracting].Io.biNegLimit:=  arrAxisCtrl[P2AxisNo.P2M3_TailCurlRetracting].Io.DigitalInputs.17;
arrAxisCtrl[P2AxisNo.P2M3_TailCurlRetracting].Io.biHomeSwitch:=arrAxisCtrl[P2AxisNo.P2M3_TailCurlRetracting].Io.DigitalInputs.17;

arrAxisCtrl[P2AxisNo.P2M3_TailCurlSEPTALine].Io.DigitalInputs;//三号叠台夹膜平移
arrAxisCtrl[P2AxisNo.P2M3_TailCurlSEPTALine].Io.biPosLimit:= arrAxisCtrl[P2AxisNo.P2M3_TailCurlSEPTALine].Io.DigitalInputs.16;
arrAxisCtrl[P2AxisNo.P2M3_TailCurlSEPTALine].Io.biNegLimit:=  arrAxisCtrl[P2AxisNo.P2M3_TailCurlSEPTALine].Io.DigitalInputs.17;
arrAxisCtrl[P2AxisNo.P2M3_TailCurlSEPTALine].Io.biHomeSwitch:=arrAxisCtrl[P2AxisNo.P2M3_TailCurlSEPTALine].Io.DigitalInputs.17;

arrAxisCtrl[P2AxisNo.P2M3_TailCurlSEPTAUpDown].Io.DigitalInputs;//三号叠台夹膜升降
arrAxisCtrl[P2AxisNo.P2M3_TailCurlSEPTAUpDown].Io.biPosLimit:= arrAxisCtrl[P2AxisNo.P2M3_TailCurlSEPTAUpDown].Io.DigitalInputs.16;
arrAxisCtrl[P2AxisNo.P2M3_TailCurlSEPTAUpDown].Io.biNegLimit:=  arrAxisCtrl[P2AxisNo.P2M3_TailCurlSEPTAUpDown].Io.DigitalInputs.2;
arrAxisCtrl[P2AxisNo.P2M3_TailCurlSEPTAUpDown].Io.biHomeSwitch:=arrAxisCtrl[P2AxisNo.P2M3_TailCurlSEPTAUpDown].Io.DigitalInputs.2;

arrAxisCtrl[P2AxisNo.P2M3_TailCurlUpDown].Io.DigitalInputs;//三号叠台尾卷夹电芯升降
arrAxisCtrl[P2AxisNo.P2M3_TailCurlUpDown].Io.biPosLimit:= arrAxisCtrl[P2AxisNo.P2M3_TailCurlUpDown].Io.DigitalInputs.16;
arrAxisCtrl[P2AxisNo.P2M3_TailCurlUpDown].Io.biNegLimit:=  arrAxisCtrl[P2AxisNo.P2M3_TailCurlUpDown].Io.DigitalInputs.17;
arrAxisCtrl[P2AxisNo.P2M3_TailCurlUpDown].Io.biHomeSwitch:=arrAxisCtrl[P2AxisNo.P2M3_TailCurlUpDown].Io.DigitalInputs.2;

arrAxisCtrl[P2AxisNo.P2M3_TailCurlWhirling].Io.DigitalInputs;//三号叠台尾卷夹电芯旋转
arrAxisCtrl[P2AxisNo.P2M3_TailCurlWhirling].Io.biPosLimit:= arrAxisCtrl[P2AxisNo.P2M3_TailCurlWhirling].Io.DigitalInputs.16;
arrAxisCtrl[P2AxisNo.P2M3_TailCurlWhirling].Io.biNegLimit:=  arrAxisCtrl[P2AxisNo.P2M3_TailCurlWhirling].Io.DigitalInputs.17;
arrAxisCtrl[P2AxisNo.P2M3_TailCurlWhirling].Io.biHomeSwitch:=arrAxisCtrl[P2AxisNo.P2M3_TailCurlWhirling].Io.DigitalInputs.17;
END_ACTION

ACTION P2_AutoLink:
//叠片系统信号
P2_sysControl.btn.System_Autonbtn;
END_ACTION

ACTION P2_InPut:
//1号叠台输入信号
P2Senser.P2M1_AnBeltsensor:=	I301[1];	//正极模切送料分段皮带1有料感应
arrCyCtrl[P2CYNo.P2M1_AnScrapbinCy].Io.DIOnSwitch:=	I301[2];	//正极片NG收纳盒伸出位
arrCyCtrl[P2CYNo.P2M1_AnScrapbinCy].Io.DIOFFSwitch:=	I301[3];	//正极片NG收纳盒缩回位
arrCyCtrl[P2EVNo.P2M1_AnCarryingVacuum].Io.DIOnSwitch:=	I301[4];	//正极送片搬运升降真空检测
arrCyCtrl[P2EVNo.P2M1_AnDTCarryingVacuum].Io.DIOnSwitch:=	I301[5];	//正极叠片搬运升降真空检测
P2M1_MachCtrl.se.AnLimitSwitch:=	I301[6];	//正极搬运防撞检测
P2Senser.P2M1_CaBeltsensor:=	I301[7];	//负极模切送料分段皮带1有料感应
arrCyCtrl[P2CYNo.P2M1_CaScrapbinCy].Io.DIOnSwitch:=	I301[8];	;//负极片NG收纳盒伸出位
arrCyCtrl[P2CYNo.P2M1_CaScrapbinCy].Io.DIOFFSwitch:=	I301[9];	//负极片NG收纳盒缩回位
arrCyCtrl[P2EVNo.P2M1_CaCarryingVacuum1].Io.DIOnSwitch:=	I301[10];	//负极送片搬运升降1真空检测
arrCyCtrl[P2EVNo.P2M1_CaCarryingVacuum2].Io.DIOnSwitch:=	I301[11];	//负极送片搬运升降2真空检测
arrCyCtrl[P2EVNo.P2M1_CaDTCarryingVacuum].Io.DIOnSwitch:=	I301[12];	//负极叠片搬运升降真空检测
P2M1_MachCtrl.se.CaLimitSwitch:=TRUE;	//I301[13];	//负极搬运防撞检测
P2Senser.P2M1_Offloadingsensor:=	I301[14];	//取料位有料感应
P2M1_MachCtrl.An_b.An_deviationCCDDone:=  I301[15];	//正极CCD纠偏定位拍照成像OK
P2M1_MachCtrl.Ca_b.Ca_deviationCCDDone:=   I301[16];	//负极CCD纠偏定位拍照成像OK
	
arrCyCtrl[P2CYNo.P2M1_PoleTapeSplicerLCy].Io.DIOnSwitch:=	I302[1];	//隔膜接带左压板气缸伸出位
arrCyCtrl[P2CYNo.P2M1_PoleTapeSplicerLCy].Io.DIOFFSwitch:=	I302[2];	//隔膜接带左压板气缸缩回位
arrCyCtrl[P2CYNo.P2M1_PoleTapeSplicerRCy].Io.DIOnSwitch:=	I302[3];	//隔膜接带右压板气缸伸出位
arrCyCtrl[P2CYNo.P2M1_PoleTapeSplicerRCy].Io.DIOFFSwitch:=	I302[4];	//隔膜接带右压板气缸缩回位
arrCyCtrl[P2CYNo.P2M1_PoleTapeCy].Io.DIOnSwitch:=	I302[5];	//隔膜夹紧气缸伸出位
arrCyCtrl[P2CYNo.P2M1_PoleTapeCy].Io.DIOFFSwitch:=	NOT I302[5];	//隔膜夹紧气缸缩回位
arrCyCtrl[P2EVNo.P2M1_AndeviationVacuum].Io.DIOnSwitch:=I302[6];//正极纠偏平台真空检测
I302[7];	//叠片平台真空检测
arrCyCtrl[P2CYNo.P2M1_PoleHotCutterCy].Io.DIOnSwitch:=	I302[8];	//隔膜热切升降伸出位
arrCyCtrl[P2CYNo.P2M1_PoleHotCutterCy].Io.DIOFFSwitch:=	I302[9];	//隔膜热切升降缩回位
P2M1_MachCtrl.btn.	PoleInflationbtn:=I302[10];	//隔膜气胀轴按钮
P2M1_MachCtrl.btn.	PoleTapeSplicerLbtn:=	I302[11];	//隔膜左压板气缸按钮
P2M1_MachCtrl.btn.	PoleTapeSplicerRbtn:=	I302[12];	//隔膜右压板气缸按钮
arrCyCtrl[P2CYNo.P2M1_PreDiaph].Io.DIOnSwitch:=	I302[13];	//压隔膜气缸伸出位
arrCyCtrl[P2CYNo.P2M1_PreDiaph].Io.DIOFFSwitch:=	I302[14];	//压隔膜气缸缩回位
arrCyCtrl[P2EVNo.P2M1_CadeviationVacuum].Io.DIOnSwitch:=	I302[15];//负极纠偏平台真空检测
P2Senser.P2M1_Yellowmark:=I302[16];	//隔膜黄标检测

arrCyCtrl[P2CYNo.P2M1_PoleSplintCy_U].Io.DIOnSwitch:=	I303[1];	//夹膜上夹板伸出位
arrCyCtrl[P2CYNo.P2M1_PoleSplintCy_U].Io.DIOFFSwitch:=	I303[2];	//夹膜上夹板缩回位
arrCyCtrl[P2CYNo.P2M1_PoleSplintCy_D].Io.DIOnSwitch:=	I303[3];	//夹膜下夹板伸出位
arrCyCtrl[P2CYNo.P2M1_PoleSplintCy_D].Io.DIOFFSwitch:=	I303[4];	//夹膜下夹板缩回位
arrCyCtrl[P2EVNo.P2M1_PoleSplintVacuum_D].Io.DIOnSwitch:=	I303[5];	//夹膜下夹板真空检测
arrCyCtrl[P2CYNo.P2M1_TailCurlSplintCy].Io.DIOnSwitch:=(TRUE AND NOT I303[7]) OR	I303[6];	//尾卷夹张开位
arrCyCtrl[P2CYNo.P2M1_TailCurlSplintCy].Io.DIOFFSwitch:=	I303[7];	//尾卷夹闭合位
arrCyCtrl[P2CYNo.P2M1_CurlingSplintCy_L].Io.DIOnSwitch:=	I303[8];	//长卷针夹张开位
arrCyCtrl[P2CYNo.P2M1_CurlingSplintCy_L].Io.DIOFFSwitch:=	I303[9];	//长卷针夹闭合位
arrCyCtrl[P2CYNo.P2M1_CurlingSplintCy_S].Io.DIOnSwitch:=	I303[10];	//短卷针夹张开位
arrCyCtrl[P2CYNo.P2M1_CurlingSplintCy_S].Io.DIOFFSwitch:=	I303[11];	//短卷针夹闭合位
arrCyCtrl[P2CYNo.P2M1_TailCurlLineCy].Io.DIOnSwitch:=	I303[12];	//尾卷压辊平移缸伸出位
arrCyCtrl[P2CYNo.P2M1_TailCurlLineCy].Io.DIOFFSwitch:=	I303[13];	//尾卷压辊平移缸缩回位
arrCyCtrl[P2CYNo.P2M1_TailCurlUpdownCy].Io.DIOnSwitch:=	I303[14];	//尾卷压辊升降缸伸出位
arrCyCtrl[P2CYNo.P2M1_TailCurlUpdownCy].Io.DIOFFSwitch:=	I303[15];	//尾卷压辊升降缸缩回位
I303[16];	//叠台CCD对检测拍成像OK
	
